KUKA KRL program: MyProgram_338().src

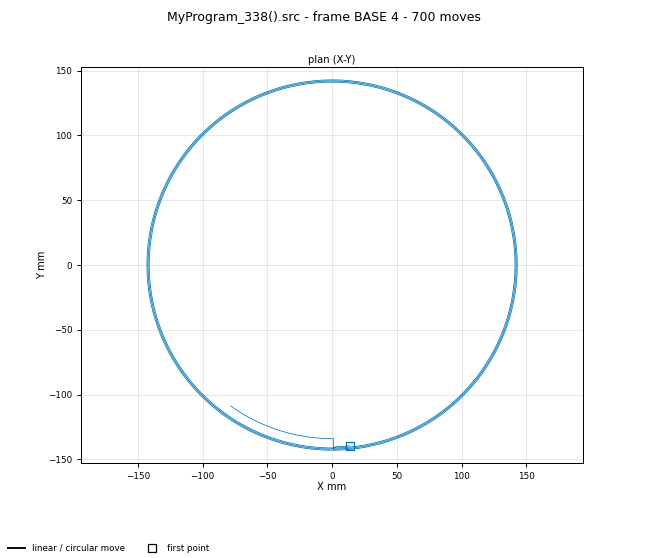
[picture p0: tool path of MyProgram_338().src in frame BASE 4, 700 of 700 moves have a stored position in this frame; points joined in program order, loops and branches not executed]
&ACCESS RVP
&REL 1
&PARAM TEMPLATE = C:\KRC\Roboter\Template\vorgabe
&PARAM EDITMASK = *
DEF MyProgram_338()
; ---- Setting reference (Base) ----
$BASE = BASE_DATA[4]

; --------------------------
; ---- Setting tool (TCP) ----
$TOOL = TOOL_DATA[3]
; --------------------------

$VEL.CP = VEL_APROX_PRINT
Startdeposition()
$VEL.CP = VEL_PRINT
LIN {X 13.5341,Y -139.6097,Z 190,A -74.3045,B 1.205,C 0.2209,E1 1.2499,E2 527.3623} C_DIS
LIN {X 10.5438,Y -139.8677,Z 190,A -75.6606,B 1.2048,C 0.2221,E1 1.246,E2 528.738} C_DIS
LIN {X 6.6617,Y -140.1064,Z 190,A -77.2712,B 1.2046,C 0.223,E1 1.2415,E2 530.3526} C_DIS
LIN {X 2.7568,Y -140.2378,Z 190,A -78.8396,B 1.2045,C 0.2236,E1 1.2371,E2 531.9178} C_DIS
LIN {X 2.7568,Y -140.2378,Z 190,A -78.8396,B 1.2045,C 0.2236,E1 1.2371,E2 531.9178} C_DIS
Enddeposition()
LIN {X 1.0179,Y -141.1573,Z 190,A -79.3498,B 1.2969,C 0.2281,E1 1.3282,E2 532.3992} C_DIS
Startdeposition()
$VEL.CP = VEL_PRINT
LIN {X 4.908,Y -141.079,Z 190,A -77.7249,B 1.297,C 0.2273,E1 1.3328,E2 530.7668} C_DIS
LIN {X 8.6277,Y -140.8992,Z 190,A -76.1602,B 1.2972,C 0.2263,E1 1.3372,E2 529.1935} C_DIS
LIN {X 12.831,Y -140.5802,Z 190,A -74.5145,B 1.2973,C 0.2256,E1 1.3418,E2 527.5564} C_DIS
LIN {X 16.4305,Y -140.2038,Z 190,A -73.2184,B 1.2973,C 0.2254,E1 1.3454,E2 526.2848} C_DIS
LIN {X 19.7873,Y -139.7694,Z 190,A -71.8875,B 1.2975,C 0.2246,E1 1.3491,E2 524.9595} C_DIS
LIN {X 23.0508,Y -139.2683,Z 190,A -70.5385,B 1.2977,C 0.2235,E1 1.3528,E2 523.6084} C_DIS
LIN {X 25.7659,Y -138.7935,Z 190,A -69.2796,B 1.298,C 0.222,E1 1.3564,E2 522.3283} C_DIS
LIN {X 31.931,Y -137.5049,Z 190,A -66.6929,B 1.2984,C 0.2195,E1 1.3635,E2 519.7355} C_DIS
LIN {X 37.4822,Y -136.0967,Z 190,A -64.7983,B 1.2984,C 0.2191,E1 1.3685,E2 517.9024} C_DIS
LIN {X 40.1642,Y -135.3293,Z 190,A -63.2039,B 1.299,C 0.2157,E1 1.3729,E2 516.2395} C_DIS
LIN {X 44.0957,Y -134.0998,Z 190,A -61.9584,B 1.299,C 0.2157,E1 1.3761,E2 515.0555} C_DIS
LIN {X 47.4169,Y -132.9615,Z 190,A -60.616,B 1.2992,C 0.2144,E1 1.3796,E2 513.7243} C_DIS
LIN {X 51.0235,Y -131.6188,Z 190,A -59.1287,B 1.2995,C 0.2128,E1 1.3835,E2 512.2467} C_DIS
LIN {X 54.9963,Y -130.0104,Z 190,A -57.4435,B 1.2998,C 0.2107,E1 1.3879,E2 510.5683} C_DIS
LIN {X 62.0576,Y -126.7908,Z 190,A -54.5002,B 1.3004,C 0.2072,E1 1.3953,E2 507.653} C_DIS
LIN {X 64.5696,Y -125.5308,Z 190,A -52.8888,B 1.301,C 0.2031,E1 1.3995,E2 505.9721} C_DIS
LIN {X 69.0352,Y -123.1325,Z 190,A -51.4052,B 1.3011,C 0.2027,E1 1.4029,E2 504.5708} C_DIS
LIN {X 72.8721,Y -120.9014,Z 190,A -49.7085,B 1.3015,C 0.2003,E1 1.407,E2 502.888} C_DIS
LIN {X 76.531,Y -118.6196,Z 190,A -48.039,B 1.3019,C 0.1977,E1 1.4109,E2 501.2289} C_DIS
LIN {X 80.3918,Y -116.0374,Z 190,A -46.2878,B 1.3023,C 0.195,E1 1.4149,E2 499.4956} C_DIS
LIN {X 84.0888,Y -113.3869,Z 190,A -44.5646,B 1.3027,C 0.1923,E1 1.4188,E2 497.789} C_DIS
LIN {X 87.6501,Y -110.6571,Z 190,A -42.8641,B 1.3031,C 0.1895,E1 1.4225,E2 496.1045} C_DIS
LIN {X 91.1163,Y -107.8213,Z 190,A -41.1614,B 1.3035,C 0.1865,E1 1.4261,E2 494.417} C_DIS
LIN {X 94.5666,Y -104.8082,Z 190,A -39.4314,B 1.304,C 0.1835,E1 1.4297,E2 492.7042} C_DIS
LIN {X 97.9221,Y -101.68,Z 190,A -37.7263,B 1.3044,C 0.1805,E1 1.4332,E2 491.0201} C_DIS
LIN {X 101.0004,Y -98.6228,Z 190,A -36.1083,B 1.3048,C 0.1775,E1 1.4363,E2 489.4213} C_DIS
LIN {X 104.054,Y -95.3951,Z 190,A -34.4823,B 1.3052,C 0.1746,E1 1.4394,E2 487.8192} C_DIS
LIN {X 106.9525,Y -92.1336,Z 190,A -32.8039,B 1.3056,C 0.1712,E1 1.4424,E2 486.1526} C_DIS
LIN {X 110.0028,Y -88.4696,Z 190,A -31.0391,B 1.3061,C 0.1677,E1 1.4455,E2 484.4107} C_DIS
LIN {X 112.8445,Y -84.8153,Z 190,A -29.3426,B 1.3065,C 0.1644,E1 1.4484,E2 482.7386} C_DIS
LIN {X 115.4716,Y -81.2022,Z 190,A -27.6775,B 1.3069,C 0.161,E1 1.451,E2 481.0931} C_DIS
LIN {X 117.9569,Y -77.5475,Z 190,A -25.997,B 1.3074,C 0.1573,E1 1.4536,E2 479.4272} C_DIS
LIN {X 122.4764,Y -70.193,Z 190,A -23.0665,B 1.308,C 0.1521,E1 1.4578,E2 476.575} C_DIS
LIN {X 124.2959,Y -66.9178,Z 190,A -21.3246,B 1.3086,C 0.1469,E1 1.4602,E2 474.8009} C_DIS
LIN {X 126.2627,Y -63.1282,Z 190,A -19.3866,B 1.3092,C 0.1413,E1 1.4626,E2 472.8327} C_DIS
LIN {X 128.4203,Y -58.6139,Z 190,A -17.927,B 1.3094,C 0.1395,E1 1.4642,E2 471.4519} C_DIS
LIN {X 129.9623,Y -55.1114,Z 190,A -16.5262,B 1.3097,C 0.1364,E1 1.4658,E2 470.0713} C_DIS
LIN {X 131.4444,Y -51.4721,Z 190,A -15.3057,B 1.3099,C 0.1345,E1 1.467,E2 468.9016} C_DIS
LIN {X 132.676,Y -48.2089,Z 190,A -14.0439,B 1.3102,C 0.1317,E1 1.4682,E2 467.6601} C_DIS
LIN {X 134.1158,Y -44.0477,Z 190,A -11.9626,B 1.3109,C 0.125,E1 1.4701,E2 465.5368} C_DIS
LIN {X 135.2678,Y -40.3742,Z 190,A -10.7965,B 1.311,C 0.1233,E1 1.471,E2 464.4246} C_DIS
LIN {X 136.1235,Y -37.3864,Z 190,A -9.4656,B 1.3114,C 0.1194,E1 1.472,E2 463.0832} C_DIS
LIN {X 136.9811,Y -34.1103,Z 190,A -8.5109,B 1.3114,C 0.1183,E1 1.4726,E2 462.1854} C_DIS
LIN {X 137.8608,Y -30.3593,Z 190,A -6.9837,B 1.3118,C 0.1142,E1 1.4735,E2 460.6622} C_DIS
LIN {X 138.5251,Y -27.17,Z 190,A -5.8094,B 1.3121,C 0.1115,E1 1.4742,E2 459.5073} C_DIS
LIN {X 139.2306,Y -23.2769,Z 190,A -4.6133,B 1.3122,C 0.1096,E1 1.4747,E2 458.3659} C_DIS
LIN {X 139.7837,Y -19.6869,Z 190,A -3.0728,B 1.3126,C 0.1051,E1 1.4754,E2 456.8155} C_DIS
LIN {X 140.3231,Y -15.3785,Z 190,A -1.5112,B 1.3129,C 0.1015,E1 1.4759,E2 455.2801} C_DIS
LIN {X 140.6221,Y -12.3552,Z 190,A -0.3436,B 1.3131,C 0.0984,E1 1.4762,E2 454.1206} C_DIS
LIN {X 140.8962,Y -8.6768,Z 190,A 0.8959,B 1.3133,C 0.0959,E1 1.4764,E2 452.915} C_DIS
LIN {X 141.0617,Y -5.3511,Z 190,A 2.2341,B 1.3136,C 0.0922,E1 1.4765,E2 451.5778} C_DIS
LIN {X 141.1597,Y -1.024,Z 190,A 3.7703,B 1.3138,C 0.0886,E1 1.4766,E2 450.0702} C_DIS
LIN {X 141.1445,Y 2.2959,Z 190,A 4.9999,B 1.314,C 0.0856,E1 1.4766,E2 448.8556} C_DIS
LIN {X 141.0255,Y 6.2803,Z 190,A 6.4937,B 1.3143,C 0.0818,E1 1.4764,E2 447.3776} C_DIS
LIN {X 140.808,Y 10.0093,Z 190,A 7.8124,B 1.3144,C 0.0788,E1 1.4762,E2 446.0843} C_DIS
LIN {X 140.52,Y 13.4588,Z 190,A 9.1794,B 1.3147,C 0.0751,E1 1.4759,E2 444.7216} C_DIS
LIN {X 140.0009,Y 18.0775,Z 190,A 10.7845,B 1.3149,C 0.0716,E1 1.4753,E2 443.1528} C_DIS
LIN {X 139.5229,Y 21.4556,Z 190,A 11.9532,B 1.3149,C 0.0691,E1 1.4749,E2 442.012} C_DIS
LIN {X 138.7901,Y 25.784,Z 190,A 13.678,B 1.3152,C 0.0645,E1 1.474,E2 440.2939} C_DIS
LIN {X 138.321,Y 28.1823,Z 190,A 15.3295,B 1.3155,C 0.0578,E1 1.4731,E2 438.5546} C_DIS
LIN {X 136.8984,Y 34.4363,Z 190,A 16.7575,B 1.3155,C 0.0578,E1 1.4722,E2 437.2804} C_DIS
LIN {X 135.2163,Y 40.5475,Z 190,A 19.3688,B 1.3158,C 0.0506,E1 1.4702,E2 434.6633} C_DIS
LIN {X 134.0733,Y 44.1752,Z 190,A 20.7118,B 1.3159,C 0.0476,E1 1.4691,E2 433.3457} C_DIS
LIN {X 132.9113,Y 47.5564,Z 190,A 22.0123,B 1.316,C 0.0446,E1 1.4679,E2 432.0642} C_DIS
LIN {X 131.6579,Y 50.9229,Z 190,A 23.21,B 1.3161,C 0.0423,E1 1.4668,E2 430.8996} C_DIS
LIN {X 130.3296,Y 54.232,Z 190,A 24.6209,B 1.3162,C 0.0387,E1 1.4653,E2 429.4928} C_DIS
LIN {X 129.1247,Y 57.0448,Z 190,A 25.9922,B 1.3163,C 0.0347,E1 1.4637,E2 428.1045} C_DIS
LIN {X 127.7624,Y 60.0367,Z 190,A 27.1031,B 1.3163,C 0.0326,E1 1.4624,E2 427.0221} C_DIS
LIN {X 126.0974,Y 63.4566,Z 190,A 28.4339,B 1.3165,C 0.0298,E1 1.4608,E2 425.718} C_DIS
LIN {X 124.1528,Y 67.1841,Z 190,A 30.0382,B 1.3165,C 0.0261,E1 1.4587,E2 424.1263} C_DIS
LIN {X 122.0248,Y 70.9752,Z 190,A 31.5717,B 1.3165,C 0.023,E1 1.4566,E2 422.6218} C_DIS
LIN {X 119.8046,Y 74.6613,Z 190,A 33.111,B 1.3167,C 0.0199,E1 1.4544,E2 421.1083} C_DIS
LIN {X 116.8635,Y 79.1857,Z 190,A 35.1623,B 1.3167,C 0.0153,E1 1.4513,E2 419.0741} C_DIS
LIN {X 114.375,Y 82.7395,Z 190,A 36.8515,B 1.3167,C 0.0115,E1 1.4486,E2 417.3937} C_DIS
LIN {X 112.1974,Y 85.6691,Z 190,A 38.4648,B 1.3167,C 0.0073,E1 1.4458,E2 415.7635} C_DIS
LIN {X 109.8202,Y 88.6959,Z 190,A 39.6553,B 1.3167,C 0.0058,E1 1.4438,E2 414.6195} C_DIS
LIN {X 106.805,Y 92.3049,Z 190,A 41.4079,B 1.3167,C 0.0023,E1 1.4406,E2 412.8862} C_DIS
LIN {X 103.7447,Y 95.7316,Z 190,A 43.1157,B 1.3168,C -0.001,E1 1.4375,E2 411.1978} C_DIS
LIN {X 100.6997,Y 98.9293,Z 190,A 44.7615,B 1.3168,C -0.0041,E1 1.4343,E2 409.5699} C_DIS
LIN {X 95.9388,Y 103.5534,Z 190,A 47.2297,B 1.3168,C -0.0085,E1 1.4294,E2 407.1295} C_DIS
LIN {X 92.6331,Y 106.5204,Z 190,A 48.9428,B 1.3168,C -0.0117,E1 1.4258,E2 405.4274} C_DIS
LIN {X 89.0531,Y 109.5313,Z 190,A 50.7172,B 1.3168,C -0.0148,E1 1.422,E2 403.6683} C_DIS
LIN {X 85.3934,Y 112.4082,Z 190,A 52.4819,B 1.3167,C -0.0178,E1 1.4181,E2 401.9189} C_DIS
LIN {X 82.8015,Y 114.33,Z 190,A 53.8155,B 1.3167,C -0.0203,E1 1.4151,E2 400.5824} C_DIS
LIN {X 78.7128,Y 117.1832,Z 190,A 55.6072,B 1.3167,C -0.0229,E1 1.411,E2 398.8192} C_DIS
LIN {X 74.8526,Y 119.6855,Z 190,A 57.3616,B 1.3166,C -0.0255,E1 1.4069,E2 397.0786} C_DIS
LIN {X 70.9387,Y 122.0459,Z 190,A 59.0952,B 1.3166,C -0.028,E1 1.4027,E2 395.3599} C_DIS
LIN {X 66.8257,Y 124.3454,Z 190,A 60.8711,B 1.3164,C -0.0305,E1 1.3984,E2 393.6007} C_DIS
LIN {X 62.3646,Y 126.6394,Z 190,A 62.6876,B 1.3164,C -0.0326,E1 1.3939,E2 391.8109} C_DIS
LIN {X 59.4283,Y 128.0437,Z 190,A 64.0461,B 1.3164,C -0.0346,E1 1.3904,E2 390.448} C_DIS
LIN {X 56.0027,Y 129.5784,Z 190,A 65.3197,B 1.3164,C -0.0357,E1 1.3872,E2 389.2048} C_DIS
LIN {X 53.4297,Y 130.6624,Z 190,A 66.6139,B 1.3163,C -0.0379,E1 1.3838,E2 387.8915} C_DIS
LIN {X 49.9777,Y 132.0203,Z 190,A 67.8219,B 1.3163,C -0.0386,E1 1.3808,E2 386.7194} C_DIS
LIN {X 46.7189,Y 133.2085,Z 190,A 69.3649,B 1.3162,C -0.0408,E1 1.3766,E2 385.1605} C_DIS
LIN {X 42.9486,Y 134.4705,Z 190,A 70.8645,B 1.3162,C -0.0422,E1 1.3727,E2 383.6749} C_DIS
LIN {X 34.9658,Y 136.764,Z 190,A 74.0337,B 1.316,C -0.045,E1 1.3642,E2 380.5308} C_DIS
LIN {X 28.4039,Y 138.2759,Z 190,A 76.722,B 1.316,C -0.0473,E1 1.3568,E2 377.8486} C_DIS
LIN {X 23.8659,Y 139.1323,Z 190,A 78.5618,B 1.3159,C -0.0487,E1 1.3517,E2 376.0135} C_DIS
LIN {X 20.457,Y 139.6737,Z 190,A 79.9473,B 1.3159,C -0.0497,E1 1.3479,E2 374.6302} C_DIS
LIN {X 16.6678,Y 140.1755,Z 190,A 81.4005,B 1.3159,C -0.0504,E1 1.3439,E2 373.1891} C_DIS
LIN {X 12.8817,Y 140.5754,Z 190,A 82.9809,B 1.3158,C -0.0514,E1 1.3394,E2 371.6052} C_DIS
LIN {X 9.1158,Y 140.8691,Z 190,A 84.4614,B 1.3158,C -0.052,E1 1.3353,E2 370.1314} C_DIS
LIN {X 5.3899,Y 141.0602,Z 190,A 85.9205,B 1.3158,C -0.0526,E1 1.3312,E2 368.6794} C_DIS
LIN {X 0.9406,Y 141.1601,Z 190,A 87.6325,B 1.3158,C -0.0529,E1 1.3264,E2 366.9792} C_DIS
LIN {X -2.4342,Y 141.1422,Z 190,A 89.0428,B 1.3158,C -0.0535,E1 1.3224,E2 365.5646} C_DIS
LIN {X -6.3851,Y 141.0204,Z 190,A 90.7043,B 1.3157,C -0.054,E1 1.3178,E2 363.8972} C_DIS
LIN {X -10.0893,Y 140.8022,Z 190,A 92.1256,B 1.3157,C -0.054,E1 1.3138,E2 362.4865} C_DIS
LIN {X -13.7127,Y 140.4956,Z 190,A 93.5119,B 1.3157,C -0.0538,E1 1.3099,E2 361.1113} C_DIS
LIN {X -18.6946,Y 139.92,Z 190,A 95.7403,B 1.3157,C -0.0543,E1 1.3037,E2 358.8611} C_DIS
LIN {X -22.8858,Y 139.2958,Z 190,A 97.3654,B 1.3157,C -0.0539,E1 1.2992,E2 357.248} C_DIS
LIN {X -26.4042,Y 138.6715,Z 190,A 98.7757,B 1.3157,C -0.0535,E1 1.2953,E2 355.8431} C_DIS
LIN {X -29.2893,Y 138.0918,Z 190,A 99.9238,B 1.3157,C -0.0531,E1 1.2921,E2 354.7011} C_DIS
LIN {X -32.6185,Y 137.3433,Z 190,A 101.2626,B 1.3157,C -0.0526,E1 1.2885,E2 353.3684} C_DIS
LIN {X -35.8886,Y 136.5254,Z 190,A 102.8458,B 1.3157,C -0.0526,E1 1.2841,E2 351.7605} C_DIS
LIN {X -39.734,Y 135.4553,Z 190,A 104.4293,B 1.3157,C -0.0518,E1 1.2798,E2 350.1822} C_DIS
LIN {X -43.1993,Y 134.3904,Z 190,A 105.9471,B 1.3158,C -0.0511,E1 1.2758,E2 348.6597} C_DIS
LIN {X -46.6395,Y 133.236,Z 190,A 107.5721,B 1.3158,C -0.0505,E1 1.2714,E2 347.0176} C_DIS
LIN {X -50.5615,Y 131.7984,Z 190,A 109.3108,B 1.3158,C -0.0494,E1 1.2668,E2 345.2747} C_DIS
LIN {X -53.7243,Y 130.5416,Z 190,A 111.0468,B 1.3158,C -0.049,E1 1.2622,E2 343.4974} C_DIS
LIN {X -57.3028,Y 129.0093,Z 190,A 112.2266,B 1.316,C -0.047,E1 1.2593,E2 342.366} C_DIS
LIN {X -59.9373,Y 127.8083,Z 190,A 113.6246,B 1.316,C -0.0463,E1 1.2556,E2 340.9422} C_DIS
LIN {X -64.8037,Y 125.4116,Z 190,A 115.9255,B 1.316,C -0.0443,E1 1.2498,E2 338.6309} C_DIS
LIN {X -67.7197,Y 123.8608,Z 190,A 117.7515,B 1.316,C -0.0436,E1 1.2452,E2 336.7476} C_DIS
LIN {X -71.9505,Y 121.4525,Z 190,A 119.3362,B 1.3162,C -0.0408,E1 1.2415,E2 335.211} C_DIS
LIN {X -75.8036,Y 119.0856,Z 190,A 121.2722,B 1.3162,C -0.0387,E1 1.2368,E2 333.2641} C_DIS
LIN {X -79.6526,Y 116.546,Z 190,A 123.5288,B 1.3162,C -0.0367,E1 1.2315,E2 330.9625} C_DIS
LIN {X -82.7587,Y 114.3611,Z 190,A 124.8474,B 1.3164,C -0.0342,E1 1.2285,E2 329.6716} C_DIS
LIN {X -86.376,Y 111.6541,Z 190,A 126.7754,B 1.3164,C -0.0316,E1 1.2242,E2 327.7335} C_DIS
LIN {X -89.8002,Y 108.9195,Z 190,A 128.7223,B 1.3164,C -0.0291,E1 1.2199,E2 325.7674} C_DIS
LIN {X -93.1849,Y 106.0386,Z 190,A 130.6176,B 1.3165,C -0.0262,E1 1.2159,E2 323.8623} C_DIS
LIN {X -96.4858,Y 103.044,Z 190,A 132.5822,B 1.3165,C -0.0233,E1 1.2118,E2 321.8801} C_DIS
LIN {X -99.7331,Y 99.9042,Z 190,A 134.5085,B 1.3166,C -0.0201,E1 1.2079,E2 319.9437} C_DIS
LIN {X -102.9011,Y 96.638,Z 190,A 136.4852,B 1.3166,C -0.0167,E1 1.2041,E2 317.9524} C_DIS
LIN {X -105.9155,Y 93.3241,Z 190,A 138.4781,B 1.3167,C -0.0133,E1 1.2003,E2 315.9393} C_DIS
LIN {X -108.8289,Y 89.9095,Z 190,A 140.4573,B 1.3167,C -0.0098,E1 1.1967,E2 313.9421} C_DIS
LIN {X -111.7395,Y 86.2659,Z 190,A 143.0809,B 1.3167,C -0.0062,E1 1.192,E2 311.2295} C_DIS
LIN {X -114.7384,Y 82.2348,Z 190,A 144.6586,B 1.3167,C -0.0017,E1 1.1895,E2 309.7105} C_DIS
LIN {X -117.6216,Y 78.0561,Z 190,A 147.0126,B 1.3167,C 0.0028,E1 1.1858,E2 307.3215} C_DIS
LIN {X -120.0757,Y 74.2256,Z 190,A 148.7681,B 1.3167,C 0.007,E1 1.1832,E2 305.5786} C_DIS
LIN {X -123.2314,Y 68.8593,Z 190,A 151.8354,B 1.3167,C 0.0127,E1 1.1788,E2 302.4458} C_DIS
LIN {X -125.2646,Y 65.0847,Z 190,A 153.7672,B 1.3167,C 0.0169,E1 1.1762,E2 300.4911} C_DIS
LIN {X -126.6424,Y 62.3585,Z 190,A 155.2188,B 1.3167,C 0.0199,E1 1.1744,E2 299.0137} C_DIS
LIN {X -129.065,Y 57.1782,Z 190,A 157.6089,B 1.3166,C 0.0256,E1 1.1716,E2 296.6165} C_DIS
LIN {X -130.8328,Y 53.0067,Z 190,A 159.3647,B 1.3165,C 0.0303,E1 1.1697,E2 294.8724} C_DIS
LIN {X -131.8984,Y 50.3033,Z 190,A 160.9161,B 1.3164,C 0.0333,E1 1.1681,E2 293.2748} C_DIS
LIN {X -133.1199,Y 46.9745,Z 190,A 162.7751,B 1.3163,C 0.037,E1 1.1663,E2 291.3631} C_DIS
LIN {X -134.4319,Y 43.0697,Z 190,A 164.4152,B 1.3161,C 0.0414,E1 1.1649,E2 289.7282} C_DIS
LIN {X -135.4564,Y 39.7301,Z 190,A 165.9508,B 1.3161,C 0.0452,E1 1.1636,E2 288.1785} C_DIS
LIN {X -136.582,Y 35.6764,Z 190,A 168.361,B 1.3159,C 0.0498,E1 1.1619,E2 285.6788} C_DIS
LIN {X -137.5372,Y 31.7898,Z 190,A 169.4919,B 1.3157,C 0.0542,E1 1.1612,E2 284.6128} C_DIS
LIN {X -138.4909,Y 27.3475,Z 190,A 171.9077,B 1.3155,C 0.0593,E1 1.1598,E2 282.1242} C_DIS
LIN {X -139.6177,Y 20.8352,Z 190,A 174.7523,B 1.3151,C 0.0667,E1 1.1584,E2 279.2601} C_DIS
LIN {X -140.2076,Y 16.3991,Z 190,A 176.7981,B 1.3148,C 0.0717,E1 1.1577,E2 277.1855} C_DIS
LIN {X -140.6293,Y 12.2697,Z 190,A 178.8072,B 1.3146,C 0.0765,E1 1.1572,E2 275.1348} C_DIS
LIN {X -141.076,Y 4.9862,Z 190,A -177.8479,B 1.3141,C 0.0848,E1 1.1567,E2 271.741} C_DIS
LIN {X -141.1544,Y -1.6978,Z 190,A -174.8323,B 1.3136,C 0.0924,E1 1.1567,E2 268.6868} C_DIS
LIN {X -141.0591,Y -5.4195,Z 190,A -172.7178,B 1.3132,C 0.0967,E1 1.1569,E2 266.4921} C_DIS
LIN {X -140.8261,Y -9.7619,Z 190,A -171.0856,B 1.3129,C 0.1016,E1 1.1572,E2 264.8788} C_DIS
LIN {X -140.2692,Y -15.8789,Z 190,A -168.3398,B 1.3123,C 0.1085,E1 1.158,E2 262.1004} C_DIS
LIN {X -139.8928,Y -18.9028,Z 190,A -166.9558,B 1.312,C 0.1119,E1 1.1585,E2 260.6971} C_DIS
LIN {X -139.0067,Y -24.5802,Z 190,A -164.4943,B 1.3115,C 0.1183,E1 1.1596,E2 258.2192} C_DIS
LIN {X -138.3734,Y -27.9252,Z 190,A -162.8143,B 1.3111,C 0.1221,E1 1.1605,E2 256.4992} C_DIS
LIN {X -137.3606,Y -32.5471,Z 190,A -160.668,B 1.3106,C 0.1273,E1 1.1619,E2 254.323} C_DIS
LIN {X -136.4058,Y -36.3372,Z 190,A -158.9309,B 1.3102,C 0.1315,E1 1.1631,E2 252.5659} C_DIS
LIN {X -135.1679,Y -40.7057,Z 190,A -156.8508,B 1.3097,C 0.1363,E1 1.1648,E2 250.4541} C_DIS
LIN {X -134.1042,Y -44.0825,Z 190,A -154.8659,B 1.3093,C 0.14,E1 1.1666,E2 248.3939} C_DIS
LIN {X -132.7877,Y -47.8992,Z 190,A -153.742,B 1.3089,C 0.1443,E1 1.1675,E2 247.342} C_DIS
LIN {X -131.7292,Y -50.7396,Z 190,A -152.1032,B 1.3085,C 0.1474,E1 1.1692,E2 245.6471} C_DIS
LIN {X -130.5921,Y -53.6035,Z 190,A -150.7696,B 1.3082,C 0.1505,E1 1.1706,E2 244.3026} C_DIS
LIN {X -128.8207,Y -57.7245,Z 190,A -148.7726,B 1.3077,C 0.155,E1 1.1729,E2 242.2815} C_DIS
LIN {X -127.435,Y -60.7225,Z 190,A -147.3619,B 1.3073,C 0.1582,E1 1.1746,E2 240.8615} C_DIS
LIN {X -125.9601,Y -63.7262,Z 190,A -145.8785,B 1.3069,C 0.1614,E1 1.1764,E2 239.361} C_DIS
LIN {X -124.2033,Y -67.09,Z 190,A -143.9513,B 1.3064,C 0.1649,E1 1.179,E2 237.3801} C_DIS
LIN {X -121.931,Y -71.1369,Z 190,A -141.8664,B 1.3059,C 0.1691,E1 1.182,E2 235.2673} C_DIS
LIN {X -119.8587,Y -74.5743,Z 190,A -140.054,B 1.3054,C 0.1727,E1 1.1847,E2 233.4295} C_DIS
LIN {X -117.3954,Y -78.3949,Z 190,A -138.1225,B 1.3049,C 0.1767,E1 1.1877,E2 231.4861} C_DIS
LIN {X -114.4747,Y -82.6019,Z 190,A -134.7109,B 1.3044,C 0.18,E1 1.1936,E2 227.8842} C_DIS
LIN {X -109.6249,Y -88.9381,Z 190,A -132.2906,B 1.3034,C 0.1873,E1 1.1976,E2 225.5822} C_DIS
LIN {X -105.789,Y -93.4672,Z 190,A -129.7053,B 1.3028,C 0.1918,E1 1.2024,E2 222.972} C_DIS
LIN {X -102.6039,Y -96.9531,Z 190,A -127.6749,B 1.3022,C 0.1952,E1 1.2063,E2 220.9255} C_DIS
LIN {X -96.4816,Y -103.048,Z 190,A -123.8603,B 1.3014,C 0.201,E1 1.214,E2 217.0669} C_DIS
LIN {X -93.118,Y -106.0973,Z 190,A -121.6916,B 1.301,C 0.2035,E1 1.2186,E2 214.8512} C_DIS
LIN {X -90.5663,Y -108.2831,Z 190,A -120.4872,B 1.3006,C 0.2059,E1 1.2212,E2 213.6699} C_DIS
LIN {X -87.1425,Y -111.0568,Z 190,A -118.5675,B 1.3002,C 0.2084,E1 1.2254,E2 211.7311} C_DIS
LIN {X -82.0556,Y -114.8665,Z 190,A -116.0908,B 1.2996,C 0.2122,E1 1.231,E2 209.2693} C_DIS
LIN {X -79.2497,Y -116.8201,Z 190,A -114.3501,B 1.2994,C 0.2134,E1 1.2351,E2 207.4773} C_DIS
LIN {X -75.223,Y -119.4527,Z 190,A -112.3535,B 1.299,C 0.2157,E1 1.2399,E2 205.4741} C_DIS
LIN {X -71.3526,Y -121.8042,Z 190,A -110.4035,B 1.2987,C 0.2176,E1 1.2446,E2 203.5075} C_DIS
LIN {X -67.4815,Y -123.9908,Z 190,A -108.3223,B 1.2985,C 0.2189,E1 1.2498,E2 201.3856} C_DIS
LIN {X -64.6281,Y -125.501,Z 190,A -107.1485,B 1.2982,C 0.2205,E1 1.2527,E2 200.2316} C_DIS
LIN {X -60.5539,Y -127.5155,Z 190,A -105.2903,B 1.2979,C 0.2221,E1 1.2574,E2 198.3711} C_DIS
LIN {X -56.7193,Y -129.2686,Z 190,A -103.4054,B 1.2978,C 0.2231,E1 1.2623,E2 196.4605} C_DIS
LIN {X -53.0407,Y -130.8191,Z 190,A -102.0121,B 1.2975,C 0.2249,E1 1.2659,E2 195.0999} C_DIS
LIN {X -49.836,Y -132.0734,Z 190,A -100.4381,B 1.2974,C 0.2254,E1 1.2701,E2 193.4997} C_DIS
LIN {X -46.557,Y -133.2646,Z 190,A -98.8487,B 1.2974,C 0.2258,E1 1.2743,E2 191.8844} C_DIS
LIN {X -39.2179,Y -135.6064,Z 190,A -95.6814,B 1.2971,C 0.2272,E1 1.2829,E2 188.7103} C_DIS
LIN {X -35.5749,Y -136.6091,Z 190,A -93.8789,B 1.2971,C 0.227,E1 1.2879,E2 186.8677} C_DIS
LIN {X -31.9044,Y -137.511,Z 190,A -92.6406,B 1.2969,C 0.2283,E1 1.2912,E2 185.6724} C_DIS
LIN {X -28.3517,Y -138.2866,Z 190,A -91.1787,B 1.2968,C 0.2287,E1 1.2952,E2 184.212} C_DIS
LIN {X -25.1026,Y -138.9132,Z 190,A -89.8389,B 1.2968,C 0.2289,E1 1.2989,E2 182.8722} C_DIS
LIN {X -21.6302,Y -139.4959,Z 190,A -88.5289,B 1.2967,C 0.2294,E1 1.3025,E2 181.5791} C_DIS
LIN {X -18.6632,Y -139.9242,Z 190,A -87.1996,B 1.2967,C 0.2291,E1 1.3062,E2 180.2328} C_DIS
LIN {X -14.6571,Y -140.4007,Z 190,A -85.4648,B 1.2967,C 0.2287,E1 1.3111,E2 178.483} C_DIS
LIN {X -10.3233,Y -140.7851,Z 190,A -83.8896,B 1.2967,C 0.2292,E1 1.3155,E2 176.9349} C_DIS
LIN {X -6.9557,Y -140.9917,Z 190,A -82.4526,B 1.2967,C 0.2287,E1 1.3195,E2 175.4874} C_DIS
LIN {X -2.8925,Y -141.1346,Z 190,A -80.7503,B 1.2969,C 0.228,E1 1.3243,E2 173.7766} C_DIS
LIN {X 1.0179,Y -141.1573,Z 190,A -79.3471,B 1.2969,C 0.2282,E1 1.3282,E2 172.3996} C_DIS
Enddeposition()
LIN {X 1.0179,Y -141.1573,Z 190,A -79.3471,B 1.2969,C 0.2282,E1 1.3282,E2 172.3996} C_DIS
Startdeposition()
$VEL.CP = VEL_PRINT
LIN {X -1.1496,Y -142.0579,Z 190,A -80.7182,B 1.2965,C 0.2309,E1 1.3242,E2 173.8709} C_DIS
LIN {X -5.1783,Y -141.968,Z 190,A -82.4266,B 1.2964,C 0.2317,E1 1.3193,E2 175.5922} C_DIS
LIN {X -9.748,Y -141.7284,Z 190,A -84.0734,B 1.2964,C 0.2313,E1 1.3148,E2 177.2107} C_DIS
LIN {X -13.0043,Y -141.4666,Z 190,A -85.5689,B 1.2964,C 0.2321,E1 1.3105,E2 178.733} C_DIS
LIN {X -16.9805,Y -141.0435,Z 190,A -87.0493,B 1.2964,C 0.2317,E1 1.3064,E2 180.1946} C_DIS
LIN {X -20.6841,Y -140.5492,Z 190,A -88.5678,B 1.2964,C 0.2317,E1 1.3022,E2 181.7155} C_DIS
LIN {X -24.3142,Y -139.9675,Z 190,A -90.2093,B 1.2964,C 0.232,E1 1.2976,E2 183.381} C_DIS
LIN {X -28.5545,Y -139.1626,Z 190,A -91.8549,B 1.2964,C 0.2314,E1 1.2931,E2 185.0132} C_DIS
LIN {X -31.8541,Y -138.4445,Z 190,A -93.1511,B 1.2965,C 0.2308,E1 1.2895,E2 186.3002} C_DIS
LIN {X -35.0471,Y -137.6707,Z 190,A -94.5933,B 1.2965,C 0.2307,E1 1.2856,E2 187.7601} C_DIS
LIN {X -39.2393,Y -136.5367,Z 190,A -96.2704,B 1.2967,C 0.2298,E1 1.281,E2 189.4268} C_DIS
LIN {X -41.7543,Y -135.787,Z 190,A -97.4715,B 1.2967,C 0.2297,E1 1.2778,E2 190.6492} C_DIS
LIN {X -47.3057,Y -133.9564,Z 190,A -99.8118,B 1.297,C 0.2283,E1 1.2715,E2 192.9878} C_DIS
LIN {X -50.2257,Y -132.8873,Z 190,A -101.1377,B 1.297,C 0.2277,E1 1.268,E2 194.3244} C_DIS
LIN {X -54.5046,Y -131.1899,Z 190,A -103.1165,B 1.2973,C 0.2266,E1 1.2628,E2 196.3215} C_DIS
LIN {X -58.4243,Y -129.4924,Z 190,A -104.8071,B 1.2975,C 0.2251,E1 1.2585,E2 198.0079} C_DIS
LIN {X -61.501,Y -128.0592,Z 190,A -106.2195,B 1.2977,C 0.224,E1 1.2549,E2 199.4269} C_DIS
LIN {X -64.7664,Y -126.4393,Z 190,A -107.745,B 1.2979,C 0.2228,E1 1.251,E2 200.9607} C_DIS
LIN {X -68.2574,Y -124.5914,Z 190,A -109.4754,B 1.2982,C 0.2214,E1 1.2467,E2 202.7113} C_DIS
LIN {X -72.2557,Y -122.3162,Z 190,A -111.4201,B 1.2985,C 0.2195,E1 1.2419,E2 204.6693} C_DIS
LIN {X -76.1205,Y -119.9492,Z 190,A -113.3207,B 1.2988,C 0.2175,E1 1.2374,E2 206.5807} C_DIS
LIN {X -79.8993,Y -117.4659,Z 190,A -115.3075,B 1.2992,C 0.2155,E1 1.2327,E2 208.5913} C_DIS
LIN {X -83.6692,Y -114.8113,Z 190,A -117.3305,B 1.2995,C 0.2132,E1 1.228,E2 210.6381} C_DIS
LIN {X -86.648,Y -112.5803,Z 190,A -118.8516,B 1.2999,C 0.2111,E1 1.2246,E2 212.1621} C_DIS
LIN {X -90.2767,Y -109.692,Z 190,A -120.8277,B 1.3003,C 0.2084,E1 1.2202,E2 214.1535} C_DIS
LIN {X -92.9319,Y -107.4512,Z 190,A -122.2922,B 1.3007,C 0.2063,E1 1.2171,E2 215.6271} C_DIS
LIN {X -96.3953,Y -104.3556,Z 190,A -124.323,B 1.3011,C 0.2034,E1 1.2128,E2 217.6804} C_DIS
LIN {X -99.5095,Y -101.3898,Z 190,A -126.3268,B 1.3015,C 0.2007,E1 1.2087,E2 219.7227} C_DIS
LIN {X -103.2802,Y -97.5461,Z 190,A -128.5035,B 1.3021,C 0.1968,E1 1.2045,E2 221.8999} C_DIS
LIN {X -106.4808,Y -94.0418,Z 190,A -130.6034,B 1.3026,C 0.1934,E1 1.2005,E2 224.0262} C_DIS
LIN {X -108.8941,Y -91.2366,Z 190,A -132.1291,B 1.3031,C 0.1905,E1 1.1977,E2 225.5563} C_DIS
LIN {X -111.4814,Y -88.0572,Z 190,A -133.9903,B 1.3035,C 0.1873,E1 1.1944,E2 227.4469} C_DIS
LIN {X -115.1699,Y -83.1743,Z 190,A -136.4044,B 1.3042,C 0.1822,E1 1.1904,E2 229.8529} C_DIS
LIN {X -117.0664,Y -80.4829,Z 190,A -138.0871,B 1.3046,C 0.1796,E1 1.1876,E2 231.5856} C_DIS
LIN {X -119.1073,Y -77.4305,Z 190,A -140.0407,B 1.305,C 0.1766,E1 1.1845,E2 233.6054} C_DIS
LIN {X -121.1645,Y -74.1702,Z 190,A -141.2379,B 1.3055,C 0.1729,E1 1.1828,E2 234.7519} C_DIS
LIN {X -122.9014,Y -71.255,Z 190,A -142.9111,B 1.3059,C 0.1699,E1 1.1804,E2 236.4676} C_DIS
LIN {X -125.065,Y -67.3856,Z 190,A -144.8827,B 1.3064,C 0.1658,E1 1.1777,E2 238.4644} C_DIS
LIN {X -126.7751,Y -64.1066,Z 190,A -146.4973,B 1.3069,C 0.1623,E1 1.1756,E2 240.0957} C_DIS
LIN {X -129.0309,Y -59.4351,Z 190,A -149.2823,B 1.3075,C 0.1575,E1 1.1722,E2 242.9762} C_DIS
LIN {X -130.8366,Y -55.3505,Z 190,A -150.6671,B 1.308,C 0.1528,E1 1.1707,E2 244.3027} C_DIS
LIN {X -131.9483,Y -52.6438,Z 190,A -152.2078,B 1.3083,C 0.15,E1 1.1691,E2 245.8929} C_DIS
LIN {X -133.3024,Y -49.1174,Z 190,A -153.7449,B 1.3088,C 0.1461,E1 1.1676,E2 247.4314} C_DIS
LIN {X -134.2463,Y -46.4696,Z 190,A -155.0726,B 1.3091,C 0.1432,E1 1.1663,E2 248.7853} C_DIS
LIN {X -135.4703,Y -42.7728,Z 190,A -156.7412,B 1.3095,C 0.1391,E1 1.1648,E2 250.4668} C_DIS
LIN {X -136.4373,Y -39.579,Z 190,A -158.2321,B 1.3099,C 0.1356,E1 1.1636,E2 251.9771} C_DIS
LIN {X -137.2762,Y -36.5619,Z 190,A -159.7143,B 1.3103,C 0.1322,E1 1.1625,E2 253.4886} C_DIS
LIN {X -138.1924,Y -32.9323,Z 190,A -161.4532,B 1.3107,C 0.1282,E1 1.1614,E2 255.2581} C_DIS
LIN {X -139.6734,Y -25.9504,Z 190,A -165.4963,B 1.3114,C 0.1204,E1 1.1591,E2 259.4568} C_DIS
LIN {X -140.672,Y -19.825,Z 190,A -167.3861,B 1.312,C 0.1135,E1 1.1584,E2 261.263} C_DIS
LIN {X -141.1693,Y -15.9162,Z 190,A -169.1057,B 1.3124,C 0.1091,E1 1.1578,E2 262.9994} C_DIS
LIN {X -141.415,Y -13.5418,Z 190,A -170.3144,B 1.3126,C 0.1064,E1 1.1574,E2 264.2406} C_DIS
LIN {X -141.8076,Y -8.5001,Z 190,A -172.5702,B 1.313,C 0.1007,E1 1.157,E2 266.5242} C_DIS
LIN {X -141.9782,Y -4.9187,Z 190,A -174.1063,B 1.3134,C 0.0967,E1 1.1568,E2 268.0715} C_DIS
LIN {X -142.0413,Y -2.4273,Z 190,A -175.3628,B 1.3136,C 0.0938,E1 1.1568,E2 269.3608} C_DIS
LIN {X -142.0359,Y 2.752,Z 190,A -177.6231,B 1.314,C 0.088,E1 1.1568,E2 271.6426} C_DIS
LIN {X -141.9405,Y 5.885,Z 190,A -179.2538,B 1.3142,C 0.0844,E1 1.157,E2 273.3208} C_DIS
LIN {X -141.6628,Y 10.6463,Z 190,A 178.6918,B 1.3145,C 0.079,E1 1.1573,E2 275.3912} C_DIS
LIN {X -141.3323,Y 14.4011,Z 190,A 177.0264,B 1.3148,C 0.0747,E1 1.1578,E2 277.0748} C_DIS
LIN {X -140.8227,Y 18.7245,Z 190,A 175.0749,B 1.3151,C 0.0699,E1 1.1585,E2 279.0506} C_DIS
LIN {X -139.8081,Y 25.2046,Z 190,A 172.1234,B 1.3154,C 0.0625,E1 1.1598,E2 282.0401} C_DIS
LIN {X -138.4993,Y 31.6144,Z 190,A 169.4501,B 1.3157,C 0.0553,E1 1.1614,E2 284.7164} C_DIS
LIN {X -136.9393,Y 37.8067,Z 190,A 166.4817,B 1.316,C 0.0484,E1 1.1634,E2 287.7338} C_DIS
LIN {X -136.1235,Y 40.6506,Z 190,A 164.988,B 1.3161,C 0.0452,E1 1.1646,E2 289.2652} C_DIS
LIN {X -135.1516,Y 43.7705,Z 190,A 163.4252,B 1.3162,C 0.0417,E1 1.166,E2 290.8583} C_DIS
LIN {X -133.9982,Y 47.1851,Z 190,A 161.9202,B 1.3164,C 0.0379,E1 1.1673,E2 292.369} C_DIS
LIN {X -132.6879,Y 50.7543,Z 190,A 160.234,B 1.3164,C 0.0339,E1 1.169,E2 294.0734} C_DIS
LIN {X -131.6998,Y 53.2604,Z 190,A 159.0272,B 1.3165,C 0.0312,E1 1.1703,E2 295.2946} C_DIS
LIN {X -130.1331,Y 56.985,Z 190,A 157.1657,B 1.3166,C 0.0271,E1 1.1724,E2 297.1843} C_DIS
LIN {X -127.2583,Y 63.1418,Z 190,A 154.1319,B 1.3167,C 0.0204,E1 1.176,E2 300.253} C_DIS
LIN {X -125.4752,Y 66.6171,Z 190,A 152.4398,B 1.3168,C 0.0166,E1 1.1782,E2 301.9586} C_DIS
LIN {X -123.2027,Y 70.734,Z 190,A 150.5002,B 1.3168,C 0.0121,E1 1.1809,E2 303.9023} C_DIS
LIN {X -120.6385,Y 75.0226,Z 190,A 148.0173,B 1.3168,C 0.0076,E1 1.1846,E2 306.4418} C_DIS
LIN {X -118.2791,Y 78.6901,Z 190,A 146.1432,B 1.3169,C 0.0037,E1 1.1874,E2 308.3289} C_DIS
LIN {X -115.8515,Y 82.2231,Z 190,A 144.0748,B 1.3169,C 0.0001,E1 1.1908,E2 310.4377} C_DIS
LIN {X -112.796,Y 86.366,Z 190,A 142.1236,B 1.3169,C -0.0044,E1 1.1941,E2 312.3721} C_DIS
LIN {X -110.642,Y 89.1088,Z 190,A 140.4129,B 1.3169,C -0.0071,E1 1.1971,E2 314.119} C_DIS
LIN {X -107.8765,Y 92.4381,Z 190,A 138.4956,B 1.3169,C -0.0105,E1 1.2006,E2 316.056} C_DIS
LIN {X -104.9021,Y 95.8007,Z 190,A 136.4987,B 1.3169,C -0.0138,E1 1.2044,E2 318.0743} C_DIS
LIN {X -101.7567,Y 99.1352,Z 190,A 134.5097,B 1.3168,C -0.0172,E1 1.2083,E2 320.079} C_DIS
LIN {X -98.5698,Y 102.3041,Z 190,A 132.589,B 1.3168,C -0.0203,E1 1.2122,E2 322.0115} C_DIS
LIN {X -95.2915,Y 105.3642,Z 190,A 130.6531,B 1.3168,C -0.0233,E1 1.2162,E2 323.9614} C_DIS
LIN {X -91.9475,Y 108.2944,Z 190,A 128.748,B 1.3166,C -0.0261,E1 1.2203,E2 325.8788} C_DIS
LIN {X -88.5557,Y 111.0852,Z 190,A 126.872,B 1.3166,C -0.0287,E1 1.2244,E2 327.766} C_DIS
LIN {X -85.0461,Y 113.7948,Z 190,A 125.0108,B 1.3166,C -0.0313,E1 1.2286,E2 329.6348} C_DIS
LIN {X -81.5246,Y 116.3439,Z 190,A 123.163,B 1.3165,C -0.0336,E1 1.2328,E2 331.4928} C_DIS
LIN {X -78.3807,Y 118.4846,Z 190,A 121.5246,B 1.3165,C -0.0355,E1 1.2367,E2 333.1425} C_DIS
LIN {X -75.0245,Y 120.6373,Z 190,A 119.8641,B 1.3164,C -0.0374,E1 1.2406,E2 334.8083} C_DIS
LIN {X -71.5323,Y 122.7409,Z 190,A 118.0833,B 1.3164,C -0.0391,E1 1.245,E2 336.6043} C_DIS
LIN {X -67.3017,Y 125.11,Z 190,A 116.0479,B 1.3163,C -0.0411,E1 1.25,E2 338.6479} C_DIS
LIN {X -63.2408,Y 127.2095,Z 190,A 114.0206,B 1.3163,C -0.0427,E1 1.2551,E2 340.6956} C_DIS
LIN {X -58.72,Y 129.3601,Z 190,A 112.1511,B 1.3161,C -0.0447,E1 1.2598,E2 342.5464} C_DIS
LIN {X -56.105,Y 130.5135,Z 190,A 110.8825,B 1.3161,C -0.0455,E1 1.2631,E2 343.8279} C_DIS
LIN {X -52.7535,Y 131.9041,Z 190,A 109.4519,B 1.3161,C -0.0467,E1 1.2668,E2 345.2538} C_DIS
LIN {X -49.4285,Y 133.1859,Z 190,A 107.9084,B 1.3161,C -0.0474,E1 1.2709,E2 346.8091} C_DIS
LIN {X -45.9771,Y 134.417,Z 190,A 106.4448,B 1.3161,C -0.0484,E1 1.2748,E2 348.2703} C_DIS
LIN {X -43.1007,Y 135.3656,Z 190,A 105.1648,B 1.316,C -0.0489,E1 1.2783,E2 349.5563} C_DIS
LIN {X -39.5769,Y 136.4379,Z 190,A 103.6802,B 1.316,C -0.0497,E1 1.2823,E2 351.0401} C_DIS
LIN {X -35.8055,Y 137.4778,Z 190,A 102.0711,B 1.316,C -0.0502,E1 1.2866,E2 352.6522} C_DIS
LIN {X -32.7492,Y 138.2365,Z 190,A 100.7037,B 1.316,C -0.0504,E1 1.2904,E2 354.0302} C_DIS
LIN {X -28.6838,Y 139.1363,Z 190,A 99.2622,B 1.3159,C -0.0515,E1 1.2943,E2 355.443} C_DIS
LIN {X -26.2871,Y 139.609,Z 190,A 98.118,B 1.3159,C -0.0513,E1 1.2975,E2 356.6055} C_DIS
LIN {X -22.3808,Y 140.2893,Z 190,A 96.554,B 1.3159,C -0.0516,E1 1.3018,E2 358.1646} C_DIS
LIN {X -19.6786,Y 140.6929,Z 190,A 95.2372,B 1.3159,C -0.0511,E1 1.3056,E2 359.506} C_DIS
LIN {X -15.4023,Y 141.2246,Z 190,A 93.7328,B 1.3159,C -0.0517,E1 1.3097,E2 360.9822} C_DIS
LIN {X -12.2953,Y 141.5293,Z 190,A 92.3044,B 1.3159,C -0.0512,E1 1.3137,E2 362.43} C_DIS
LIN {X -7.9795,Y 141.8397,Z 190,A 90.6513,B 1.3159,C -0.0512,E1 1.3184,E2 364.0716} C_DIS
LIN {X -4.1639,Y 142.0011,Z 190,A 89.0686,B 1.3159,C -0.0507,E1 1.3228,E2 365.6586} C_DIS
LIN {X -0.6532,Y 142.0606,Z 190,A 87.7263,B 1.3159,C -0.0505,E1 1.3266,E2 366.9917} C_DIS
LIN {X 3.2443,Y 142.0267,Z 190,A 86.2228,B 1.3159,C -0.0501,E1 1.3308,E2 368.4867} C_DIS
LIN {X 6.2401,Y 141.9266,Z 190,A 84.9999,B 1.3159,C -0.0495,E1 1.3342,E2 369.7108} C_DIS
LIN {X 9.1747,Y 141.7661,Z 190,A 83.8408,B 1.3159,C -0.049,E1 1.3375,E2 370.8663} C_DIS
LIN {X 12.2602,Y 141.5322,Z 190,A 82.6139,B 1.316,C -0.0484,E1 1.3409,E2 372.0903} C_DIS
LIN {X 15.8077,Y 141.181,Z 190,A 81.2025,B 1.316,C -0.0476,E1 1.3448,E2 373.4981} C_DIS
LIN {X 19.3167,Y 140.7446,Z 190,A 79.6676,B 1.316,C -0.0463,E1 1.3491,E2 375.0454} C_DIS
LIN {X 23.4979,Y 140.105,Z 190,A 78.0441,B 1.3161,C -0.0453,E1 1.3536,E2 376.6585} C_DIS
LIN {X 27.109,Y 139.4519,Z 190,A 76.7527,B 1.3161,C -0.0447,E1 1.3571,E2 377.9273} C_DIS
LIN {X 29.7541,Y 138.9111,Z 190,A 75.565,B 1.3161,C -0.0434,E1 1.3604,E2 379.1265} C_DIS
LIN {X 33.8151,Y 137.9796,Z 190,A 74.017,B 1.3162,C -0.0423,E1 1.3646,E2 380.6584} C_DIS
LIN {X 36.8127,Y 137.2093,Z 190,A 72.7544,B 1.3162,C -0.041,E1 1.368,E2 381.9224} C_DIS
LIN {X 40.3404,Y 136.2143,Z 190,A 71.0738,B 1.3163,C -0.0386,E1 1.3726,E2 383.6265} C_DIS
LIN {X 44.0074,Y 135.0759,Z 190,A 69.9387,B 1.3163,C -0.0385,E1 1.3755,E2 384.7125} C_DIS
LIN {X 47.1297,Y 134.0174,Z 190,A 68.6827,B 1.3163,C -0.0372,E1 1.3789,E2 385.9594} C_DIS
LIN {X 50.042,Y 132.9561,Z 190,A 67.4439,B 1.3164,C -0.0357,E1 1.3821,E2 387.1966} C_DIS
LIN {X 54.1034,Y 131.3574,Z 190,A 65.8028,B 1.3164,C -0.0339,E1 1.3864,E2 388.8232} C_DIS
LIN {X 57.0871,Y 130.0889,Z 190,A 64.5512,B 1.3165,C -0.0323,E1 1.3896,E2 390.068} C_DIS
LIN {X 59.9371,Y 128.7987,Z 190,A 63.3161,B 1.3165,C -0.0306,E1 1.3927,E2 391.2996} C_DIS
LIN {X 64.0593,Y 126.7992,Z 190,A 61.5274,B 1.3166,C -0.0281,E1 1.3972,E2 393.081} C_DIS
LIN {X 67.7379,Y 124.8748,Z 190,A 59.9115,B 1.3166,C -0.0258,E1 1.4012,E2 394.6898} C_DIS
LIN {X 71.8465,Y 122.5566,Z 190,A 58.198,B 1.3166,C -0.0235,E1 1.4053,E2 396.3804} C_DIS
LIN {X 75.0768,Y 120.6048,Z 190,A 56.7116,B 1.3167,C -0.0211,E1 1.4088,E2 397.8623} C_DIS
LIN {X 78.7534,Y 118.2369,Z 190,A 55.1972,B 1.3167,C -0.0192,E1 1.4123,E2 399.3465} C_DIS
LIN {X 82.0273,Y 115.9896,Z 190,A 53.6191,B 1.3168,C -0.0164,E1 1.4159,E2 400.9218} C_DIS
LIN {X 85.0452,Y 113.7955,Z 190,A 52.2059,B 1.3168,C -0.0141,E1 1.4191,E2 402.3239} C_DIS
LIN {X 88.3846,Y 111.2214,Z 190,A 50.6093,B 1.3168,C -0.0113,E1 1.4226,E2 403.9078} C_DIS
LIN {X 91.5838,Y 108.6027,Z 190,A 49.075,B 1.3168,C -0.0087,E1 1.4259,E2 405.426} C_DIS
LIN {X 94.6364,Y 105.9529,Z 190,A 47.5519,B 1.3168,C -0.006,E1 1.4291,E2 406.936} C_DIS
LIN {X 97.7531,Y 103.0849,Z 190,A 45.8624,B 1.3169,C -0.0025,E1 1.4325,E2 408.6233} C_DIS
LIN {X 100.5029,Y 100.4059,Z 190,A 44.4785,B 1.3169,C -0.0001,E1 1.4352,E2 409.9871} C_DIS
LIN {X 103.7485,Y 97.0483,Z 190,A 42.7679,B 1.3169,C 0.0031,E1 1.4385,E2 411.6766} C_DIS
LIN {X 106.6504,Y 93.85,Z 190,A 41.2239,B 1.3169,C 0.0059,E1 1.4413,E2 413.1964} C_DIS
LIN {X 109.2614,Y 90.7966,Z 190,A 39.7193,B 1.3169,C 0.009,E1 1.444,E2 414.6869} C_DIS
LIN {X 111.7886,Y 87.6661,Z 190,A 38.1863,B 1.3169,C 0.0122,E1 1.4467,E2 416.209} C_DIS
LIN {X 114.5949,Y 83.9647,Z 190,A 36.4939,B 1.3169,C 0.0156,E1 1.4495,E2 417.8792} C_DIS
LIN {X 117.1185,Y 80.4069,Z 190,A 34.8751,B 1.3168,C 0.0191,E1 1.452,E2 419.4807} C_DIS
LIN {X 119.6719,Y 76.5549,Z 190,A 33.2888,B 1.3168,C 0.022,E1 1.4544,E2 421.0325} C_DIS
LIN {X 121.6958,Y 73.2955,Z 190,A 31.7429,B 1.3167,C 0.0259,E1 1.4567,E2 422.5787} C_DIS
LIN {X 123.9564,Y 69.404,Z 190,A 30.0935,B 1.3166,C 0.0295,E1 1.4589,E2 424.2076} C_DIS
LIN {X 126.1196,Y 65.3899,Z 190,A 28.4724,B 1.3165,C 0.0329,E1 1.461,E2 425.8015} C_DIS
LIN {X 127.7573,Y 62.1302,Z 190,A 27.1479,B 1.3165,C 0.0358,E1 1.4626,E2 427.1078} C_DIS
LIN {X 129.0983,Y 59.2893,Z 190,A 25.9665,B 1.3163,C 0.0386,E1 1.464,E2 428.2786} C_DIS
LIN {X 130.5332,Y 56.0595,Z 190,A 24.7114,B 1.3163,C 0.0413,E1 1.4654,E2 429.5124} C_DIS
LIN {X 131.7845,Y 53.0503,Z 190,A 23.4513,B 1.3162,C 0.0444,E1 1.4667,E2 430.7659} C_DIS
LIN {X 133.3538,Y 48.9793,Z 190,A 21.9082,B 1.316,C 0.0478,E1 1.4682,E2 432.2819} C_DIS
LIN {X 134.3249,Y 46.243,Z 190,A 20.8255,B 1.316,C 0.0504,E1 1.4692,E2 433.3536} C_DIS
LIN {X 135.5608,Y 42.4896,Z 190,A 19.1221,B 1.3157,C 0.0554,E1 1.4707,E2 435.0718} C_DIS
LIN {X 136.54,Y 39.2282,Z 190,A 18.1728,B 1.3157,C 0.0566,E1 1.4714,E2 435.9668} C_DIS
LIN {X 137.3638,Y 36.2333,Z 190,A 16.9274,B 1.3155,C 0.0599,E1 1.4723,E2 437.2118} C_DIS
LIN {X 138.437,Y 31.8873,Z 190,A 15.1556,B 1.3153,C 0.0647,E1 1.4734,E2 438.98} C_DIS
LIN {X 139.3452,Y 27.657,Z 190,A 13.6541,B 1.3151,C 0.068,E1 1.4742,E2 440.4506} C_DIS
LIN {X 140.1767,Y 23.0686,Z 190,A 12.0114,B 1.3149,C 0.0718,E1 1.475,E2 442.0629} C_DIS
LIN {X 140.7499,Y 19.2798,Z 190,A 10.7142,B 1.3148,C 0.0745,E1 1.4755,E2 443.3284} C_DIS
LIN {X 141.0888,Y 16.6008,Z 190,A 9.7531,B 1.3147,C 0.0768,E1 1.4758,E2 444.273} C_DIS
LIN {X 141.4156,Y 13.5356,Z 190,A 8.5909,B 1.3145,C 0.0797,E1 1.4761,E2 445.4251} C_DIS
LIN {X 141.7147,Y 9.9358,Z 190,A 7.286,B 1.3143,C 0.0829,E1 1.4764,E2 446.7107} C_DIS
LIN {X 141.8934,Y 6.9222,Z 190,A 6.1834,B 1.3141,C 0.0855,E1 1.4766,E2 447.7987} C_DIS
LIN {X 142.0129,Y 3.7423,Z 190,A 5.0211,B 1.3139,C 0.0884,E1 1.4766,E2 448.9455} C_DIS
LIN {X 142.0625,Y -0.3146,Z 190,A 3.4828,B 1.3137,C 0.0924,E1 1.4767,E2 450.4716} C_DIS
LIN {X 142.0045,Y -4.0431,Z 190,A 2.1804,B 1.3135,C 0.0953,E1 1.4767,E2 451.7478} C_DIS
LIN {X 141.8409,Y -7.9601,Z 190,A 0.6141,B 1.3131,C 0.0996,E1 1.4764,E2 453.3133} C_DIS
LIN {X 141.5765,Y -11.7356,Z 190,A -0.7152,B 1.3129,C 0.1027,E1 1.4761,E2 454.6169} C_DIS
LIN {X 141.1096,Y -16.4261,Z 190,A -2.4266,B 1.3126,C 0.1068,E1 1.4756,E2 456.3039} C_DIS
LIN {X 140.5775,Y -20.486,Z 190,A -3.9544,B 1.3123,C 0.1106,E1 1.4751,E2 457.816} C_DIS
LIN {X 139.982,Y -24.2328,Z 190,A -5.2161,B 1.312,C 0.1132,E1 1.4745,E2 459.0423} C_DIS
LIN {X 139.487,Y -26.9258,Z 190,A -6.1863,B 1.3118,C 0.1154,E1 1.474,E2 459.9949} C_DIS
LIN {X 138.9366,Y -29.6358,Z 190,A -7.1608,B 1.3116,C 0.1176,E1 1.4735,E2 460.9509} C_DIS
LIN {X 138.3205,Y -32.397,Z 190,A -8.4072,B 1.3113,C 0.1214,E1 1.4727,E2 462.2125} C_DIS
LIN {X 137.0674,Y -37.3433,Z 190,A -10.1109,B 1.311,C 0.1248,E1 1.4715,E2 463.8691} C_DIS
LIN {X 136.3075,Y -40.0222,Z 190,A -11.9567,B 1.3102,C 0.1323,E1 1.47,E2 465.8143} C_DIS
LIN {X 134.2569,Y -46.4391,Z 190,A -13.384,B 1.3103,C 0.1316,E1 1.4689,E2 467.0667} C_DIS
LIN {X 132.648,Y -50.8568,Z 190,A -15.2853,B 1.3098,C 0.1367,E1 1.467,E2 468.9701} C_DIS
LIN {X 131.2839,Y -54.2795,Z 190,A -16.7916,B 1.3094,C 0.1407,E1 1.4654,E2 470.4804} C_DIS
LIN {X 129.6292,Y -58.1184,Z 190,A -18.195,B 1.3091,C 0.1434,E1 1.4639,E2 471.8456} C_DIS
LIN {X 127.5683,Y -62.5134,Z 190,A -19.8626,B 1.3087,C 0.1467,E1 1.462,E2 473.4743} C_DIS
LIN {X 125.8274,Y -65.9464,Z 190,A -21.4439,B 1.3082,C 0.1508,E1 1.4599,E2 475.0607} C_DIS
LIN {X 123.8175,Y -69.651,Z 190,A -23.3321,B 1.3076,C 0.1562,E1 1.4573,E2 476.9766} C_DIS
LIN {X 121.8509,Y -73.0374,Z 190,A -24.598,B 1.3074,C 0.1583,E1 1.4556,E2 478.1998} C_DIS
LIN {X 119.9569,Y -76.1083,Z 190,A -25.8389,B 1.3071,C 0.1606,E1 1.4538,E2 479.4118} C_DIS
LIN {X 117.6012,Y -79.6994,Z 190,A -27.4315,B 1.3067,C 0.1639,E1 1.4513,E2 480.9861} C_DIS
LIN {X 114.9904,Y -83.4221,Z 190,A -29.0964,B 1.3062,C 0.1673,E1 1.4487,E2 482.6285} C_DIS
LIN {X 112.3499,Y -86.9456,Z 190,A -30.7462,B 1.3058,C 0.1707,E1 1.4459,E2 484.2618} C_DIS
LIN {X 109.5026,Y -90.5053,Z 190,A -32.4522,B 1.3053,C 0.1741,E1 1.4429,E2 485.9505} C_DIS
LIN {X 106.3725,Y -94.1643,Z 190,A -34.2401,B 1.3049,C 0.1776,E1 1.4397,E2 487.7179} C_DIS
LIN {X 103.214,Y -97.6162,Z 190,A -35.9699,B 1.3044,C 0.1808,E1 1.4364,E2 489.4268} C_DIS
LIN {X 99.9038,Y -101.0018,Z 190,A -37.739,B 1.304,C 0.1841,E1 1.4329,E2 491.1773} C_DIS
LIN {X 96.4945,Y -104.2642,Z 190,A -39.5096,B 1.3035,C 0.1873,E1 1.4294,E2 492.9305} C_DIS
LIN {X 93.0089,Y -107.3849,Z 190,A -41.2728,B 1.3031,C 0.1904,E1 1.4257,E2 494.6774} C_DIS
LIN {X 89.4644,Y -110.3552,Z 190,A -43.0152,B 1.3026,C 0.1934,E1 1.422,E2 496.4036} C_DIS
LIN {X 85.7344,Y -113.277,Z 190,A -44.7592,B 1.3022,C 0.1961,E1 1.4181,E2 498.125} C_DIS
LIN {X 82.3296,Y -115.7756,Z 190,A -46.3665,B 1.3018,C 0.1987,E1 1.4145,E2 499.7198} C_DIS
LIN {X 78.6335,Y -118.3169,Z 190,A -48.0288,B 1.3014,C 0.2012,E1 1.4107,E2 501.3623} C_DIS
LIN {X 74.961,Y -120.6768,Z 190,A -49.7128,B 1.301,C 0.2038,E1 1.4067,E2 503.0365} C_DIS
LIN {X 70.9119,Y -123.1,Z 190,A -51.5226,B 1.3006,C 0.2065,E1 1.4024,E2 504.8343} C_DIS
LIN {X 65.9222,Y -125.8401,Z 190,A -53.6171,B 1.3002,C 0.2091,E1 1.3973,E2 506.9011} C_DIS
LIN {X 62.3025,Y -127.6723,Z 190,A -55.1998,B 1.2999,C 0.2112,E1 1.3933,E2 508.4773} C_DIS
LIN {X 58.2476,Y -129.5714,Z 190,A -57.1834,B 1.2993,C 0.2147,E1 1.3882,E2 510.4879} C_DIS
LIN {X 54.7488,Y -131.0879,Z 190,A -58.3473,B 1.2993,C 0.215,E1 1.3853,E2 511.5985} C_DIS
LIN {X 51.3432,Y -132.4589,Z 190,A -59.7083,B 1.299,C 0.2163,E1 1.3818,E2 512.9431} C_DIS
LIN {X 48.3358,Y -133.5858,Z 190,A -60.9787,B 1.2988,C 0.2178,E1 1.3784,E2 514.2107} C_DIS
LIN {X 44.4695,Y -134.9227,Z 190,A -62.8372,B 1.2983,C 0.2207,E1 1.3734,E2 516.1009} C_DIS
LIN {X 40.9608,Y -136.0299,Z 190,A -63.9284,B 1.2983,C 0.2207,E1 1.3706,E2 517.1358} C_DIS
LIN {X 37.431,Y -137.0443,Z 190,A -65.3616,B 1.2981,C 0.222,E1 1.3668,E2 518.5629} C_DIS
LIN {X 34.3033,Y -137.8595,Z 190,A -66.6946,B 1.2978,C 0.2234,E1 1.3631,E2 519.9011} C_DIS
LIN {X 25.9667,Y -139.6703,Z 190,A -69.9351,B 1.2974,C 0.2256,E1 1.3543,E2 523.1145} C_DIS
LIN {X 22.8819,Y -140.2078,Z 190,A -71.147,B 1.2974,C 0.2264,E1 1.3509,E2 524.3196} C_DIS
LIN {X 19.6762,Y -140.6933,Z 190,A -72.5577,B 1.2971,C 0.2278,E1 1.347,E2 525.7462} C_DIS
LIN {X 15.6321,Y -141.1999,Z 190,A -74.1564,B 1.2969,C 0.2287,E1 1.3425,E2 527.3392} C_DIS
LIN {X 11.802,Y -141.5709,Z 190,A -75.5939,B 1.2969,C 0.2291,E1 1.3385,E2 528.7608} C_DIS
LIN {X 7.4805,Y -141.8653,Z 190,A -77.287,B 1.2967,C 0.2298,E1 1.3338,E2 530.447} C_DIS
LIN {X 4.2105,Y -141.9999,Z 190,A -78.5439,B 1.2967,C 0.2301,E1 1.3303,E2 531.6953} C_DIS
LIN {X 1.0282,Y -142.0561,Z 190,A -79.3363,B 1.2969,C 0.2288,E1 1.3283,E2 532.4159} C_DIS
Enddeposition()
LIN {X 1.0282,Y -142.0561,Z 190,A -79.3365,B 1.2969,C 0.2288,E1 1.3283,E2 532.416} C_DIS
Startdeposition()
$VEL.CP = VEL_PRINT
LIN {X 1.7616,Y -142.9514,Z 190,A -78.9154,B 1.2968,C 0.2288,E1 1.3293,E2 532.0023} C_DIS
LIN {X 5.2668,Y -142.8642,Z 190,A -77.5034,B 1.2968,C 0.2282,E1 1.3333,E2 530.5885} C_DIS
LIN {X 8.7679,Y -142.6917,Z 190,A -76.1725,B 1.2969,C 0.2278,E1 1.337,E2 529.2679} C_DIS
LIN {X 12.2835,Y -142.4323,Z 190,A -74.7749,B 1.2971,C 0.227,E1 1.3409,E2 527.8718} C_DIS
LIN {X 15.9944,Y -142.065,Z 190,A -73.3439,B 1.2971,C 0.2263,E1 1.3449,E2 526.4495} C_DIS
LIN {X 19.2469,Y -141.6608,Z 190,A -72.0619,B 1.2973,C 0.2256,E1 1.3485,E2 525.1714} C_DIS
LIN {X 22.7131,Y -141.1473,Z 190,A -70.6119,B 1.2975,C 0.2243,E1 1.3525,E2 523.7137} C_DIS
LIN {X 26.2114,Y -140.5387,Z 190,A -69.2975,B 1.2977,C 0.2236,E1 1.3561,E2 522.4146} C_DIS
LIN {X 29.6475,Y -139.8537,Z 190,A -67.9426,B 1.2978,C 0.2226,E1 1.3598,E2 521.0662} C_DIS
LIN {X 33.0597,Y -139.0863,Z 190,A -66.592,B 1.298,C 0.2215,E1 1.3635,E2 519.7223} C_DIS
LIN {X 36.4471,Y -138.2371,Z 190,A -65.2455,B 1.2982,C 0.2203,E1 1.3671,E2 518.3828} C_DIS
LIN {X 39.8102,Y -137.3062,Z 190,A -63.8543,B 1.2985,C 0.2189,E1 1.3709,E2 516.9918} C_DIS
LIN {X 43.9179,Y -136.0482,Z 190,A -62.2273,B 1.2987,C 0.2173,E1 1.3752,E2 515.3777} C_DIS
LIN {X 48.3801,Y -134.5253,Z 190,A -60.4948,B 1.299,C 0.2158,E1 1.3798,E2 513.6673} C_DIS
LIN {X 51.4502,Y -133.3818,Z 190,A -59.1917,B 1.2993,C 0.2142,E1 1.3832,E2 512.3647} C_DIS
LIN {X 54.742,Y -132.0649,Z 190,A -57.7945,B 1.2995,C 0.2124,E1 1.3868,E2 510.9701} C_DIS
LIN {X 58.7565,Y -130.3285,Z 190,A -56.0688,B 1.2999,C 0.2101,E1 1.3912,E2 509.2472} C_DIS
LIN {X 62.8154,Y -128.4216,Z 190,A -54.4234,B 1.3002,C 0.2082,E1 1.3953,E2 507.623} C_DIS
LIN {X 65.8362,Y -126.9005,Z 190,A -53.1013,B 1.3005,C 0.2063,E1 1.3986,E2 506.3049} C_DIS
LIN {X 69.7096,Y -124.8157,Z 190,A -51.5082,B 1.3008,C 0.2044,E1 1.4025,E2 504.7356} C_DIS
LIN {X 73.4033,Y -122.6795,Z 190,A -49.8919,B 1.3012,C 0.2021,E1 1.4064,E2 503.1318} C_DIS
LIN {X 76.4857,Y -120.7817,Z 190,A -48.5416,B 1.3015,C 0.2001,E1 1.4096,E2 501.7952} C_DIS
LIN {X 80.0557,Y -118.4455,Z 190,A -46.9371,B 1.3019,C 0.1977,E1 1.4133,E2 500.2049} C_DIS
LIN {X 83.2845,Y -116.1979,Z 190,A -45.3912,B 1.3023,C 0.195,E1 1.4168,E2 498.6623} C_DIS
LIN {X 86.8112,Y -113.5872,Z 190,A -43.7603,B 1.3027,C 0.1923,E1 1.4204,E2 497.0489} C_DIS
LIN {X 90.0149,Y -111.066,Z 190,A -42.3125,B 1.303,C 0.1902,E1 1.4235,E2 495.627} C_DIS
LIN {X 92.7983,Y -108.751,Z 190,A -40.8599,B 1.3034,C 0.1873,E1 1.4266,E2 494.1731} C_DIS
LIN {X 96.0963,Y -105.8477,Z 190,A -39.3541,B 1.3037,C 0.1852,E1 1.4297,E2 492.7031} C_DIS
LIN {X 98.6633,Y -103.4592,Z 190,A -37.9359,B 1.3041,C 0.1822,E1 1.4326,E2 491.282} C_DIS
LIN {X 101.7889,Y -100.3863,Z 190,A -36.2925,B 1.3046,C 0.1791,E1 1.4358,E2 489.6537} C_DIS
LIN {X 104.7395,Y -97.3031,Z 190,A -34.8057,B 1.3049,C 0.1767,E1 1.4386,E2 488.1981} C_DIS
LIN {X 107.1781,Y -94.6103,Z 190,A -33.3612,B 1.3053,C 0.1735,E1 1.4413,E2 486.7541} C_DIS
LIN {X 110.0275,Y -91.2809,Z 190,A -31.8672,B 1.3056,C 0.1711,E1 1.444,E2 485.2967} C_DIS
LIN {X 112.6328,Y -88.0466,Z 190,A -30.3012,B 1.3061,C 0.1678,E1 1.4467,E2 483.7437} C_DIS
LIN {X 115.2871,Y -84.5407,Z 190,A -28.6974,B 1.3065,C 0.1646,E1 1.4493,E2 482.1614} C_DIS
LIN {X 117.4557,Y -81.501,Z 190,A -27.3405,B 1.3068,C 0.1619,E1 1.4515,E2 480.8233} C_DIS
LIN {X 119.7729,Y -78.0561,Z 190,A -25.7988,B 1.3072,C 0.1586,E1 1.4538,E2 479.2979} C_DIS
LIN {X 121.7928,Y -74.865,Z 190,A -24.4362,B 1.3075,C 0.1558,E1 1.4558,E2 477.9558} C_DIS
LIN {X 123.9123,Y -71.3031,Z 190,A -22.9009,B 1.3079,C 0.1524,E1 1.4579,E2 476.4372} C_DIS
LIN {X 125.7282,Y -68.0504,Z 190,A -21.4818,B 1.3083,C 0.1491,E1 1.4598,E2 475.0275} C_DIS
LIN {X 127.3003,Y -65.0564,Z 190,A -20.3208,B 1.3086,C 0.1468,E1 1.4613,E2 473.8932} C_DIS
LIN {X 128.8501,Y -61.9309,Z 190,A -19.039,B 1.3089,C 0.144,E1 1.4629,E2 472.6269} C_DIS
LIN {X 130.3857,Y -58.6285,Z 190,A -17.627,B 1.3093,C 0.1405,E1 1.4645,E2 471.2205} C_DIS
LIN {X 132.1685,Y -54.4939,Z 190,A -16.068,B 1.3096,C 0.1373,E1 1.4661,E2 469.695} C_DIS
LIN {X 133.4648,Y -51.2367,Z 190,A -14.8058,B 1.3099,C 0.1344,E1 1.4674,E2 468.4519} C_DIS
LIN {X 134.6028,Y -48.1652,Z 190,A -13.5925,B 1.3102,C 0.1316,E1 1.4686,E2 467.2516} C_DIS
LIN {X 135.7698,Y -44.771,Z 190,A -12.2967,B 1.3105,C 0.1286,E1 1.4697,E2 465.9748} C_DIS
LIN {X 137.0283,Y -40.7594,Z 190,A -10.7017,B 1.3109,C 0.1246,E1 1.471,E2 464.3914} C_DIS
LIN {X 137.8736,Y -37.8035,Z 190,A -9.6548,B 1.3111,C 0.1224,E1 1.4717,E2 463.3695} C_DIS
LIN {X 138.7365,Y -34.5021,Z 190,A -8.4138,B 1.3114,C 0.1195,E1 1.4726,E2 462.1452} C_DIS
LIN {X 139.5407,Y -31.0917,Z 190,A -7.1437,B 1.3116,C 0.1165,E1 1.4734,E2 460.8929} C_DIS
LIN {X 140.2613,Y -27.6625,Z 190,A -5.8703,B 1.3119,C 0.1134,E1 1.4741,E2 459.6367} C_DIS
LIN {X 140.8965,Y -24.2162,Z 190,A -4.585,B 1.3122,C 0.1103,E1 1.4747,E2 458.367} C_DIS
LIN {X 141.4469,Y -20.7563,Z 190,A -3.3712,B 1.3124,C 0.1076,E1 1.4752,E2 457.1786} C_DIS
LIN {X 141.8877,Y -17.4921,Z 190,A -2.1192,B 1.3126,C 0.1044,E1 1.4756,E2 455.9352} C_DIS
LIN {X 142.2951,Y -13.7803,Z 190,A -0.7739,B 1.3129,C 0.1011,E1 1.476,E2 454.6097} C_DIS
LIN {X 142.5902,Y -10.2882,Z 190,A 0.4607,B 1.3131,C 0.0983,E1 1.4763,E2 453.3976} C_DIS
LIN {X 142.8001,Y -6.7894,Z 190,A 1.7538,B 1.3133,C 0.0951,E1 1.4765,E2 452.1189} C_DIS
LIN {X 142.925,Y -3.2785,Z 190,A 3.0509,B 1.3136,C 0.0918,E1 1.4765,E2 450.8361} C_DIS
LIN {X 142.963,Y -0.0021,Z 190,A 4.3569,B 1.3138,C 0.0882,E1 1.4765,E2 449.5305} C_DIS
LIN {X 142.9185,Y 3.5106,Z 190,A 5.5106,B 1.314,C 0.0858,E1 1.4765,E2 448.4105} C_DIS
LIN {X 142.7774,Y 7.2416,Z 190,A 6.8173,B 1.3142,C 0.0828,E1 1.4764,E2 447.1286} C_DIS
LIN {X 142.5554,Y 10.7652,Z 190,A 8.1029,B 1.3144,C 0.0797,E1 1.4761,E2 445.8598} C_DIS
LIN {X 142.2503,Y 14.2478,Z 190,A 9.3871,B 1.3146,C 0.0765,E1 1.4758,E2 444.5907} C_DIS
LIN {X 141.8593,Y 17.7302,Z 190,A 10.6544,B 1.3147,C 0.0735,E1 1.4754,E2 443.3411} C_DIS
LIN {X 141.4155,Y 20.976,Z 190,A 11.8496,B 1.3149,C 0.0706,E1 1.4749,E2 442.1611} C_DIS
LIN {X 140.8166,Y 24.6722,Z 190,A 13.1593,B 1.315,C 0.0676,E1 1.4743,E2 440.8761} C_DIS
LIN {X 140.209,Y 27.92,Z 190,A 14.4186,B 1.3152,C 0.0643,E1 1.4737,E2 439.6249} C_DIS
LIN {X 139.4846,Y 31.3376,Z 190,A 15.7667,B 1.3154,C 0.0608,E1 1.4729,E2 438.2831} C_DIS
LIN {X 138.6767,Y 34.7374,Z 190,A 16.9528,B 1.3154,C 0.0583,E1 1.4721,E2 437.125} C_DIS
LIN {X 137.7863,Y 38.1156,Z 190,A 18.2206,B 1.3156,C 0.0553,E1 1.4712,E2 435.8741} C_DIS
LIN {X 136.7199,Y 41.7776,Z 190,A 19.5961,B 1.3158,C 0.0521,E1 1.4701,E2 434.5182} C_DIS
LIN {X 135.6738,Y 45.0593,Z 190,A 20.9586,B 1.3158,C 0.0485,E1 1.4689,E2 433.1575} C_DIS
LIN {X 134.0002,Y 49.8171,Z 190,A 22.6934,B 1.316,C 0.0448,E1 1.4673,E2 431.4597} C_DIS
LIN {X 132.739,Y 53.0867,Z 190,A 24.0161,B 1.3161,C 0.0416,E1 1.466,E2 430.1471} C_DIS
LIN {X 131.3069,Y 56.535,Z 190,A 25.2792,B 1.3162,C 0.039,E1 1.4646,E2 428.9141} C_DIS
LIN {X 129.9252,Y 59.6428,Z 190,A 26.5808,B 1.3162,C 0.0358,E1 1.4631,E2 427.62} C_DIS
LIN {X 128.4264,Y 62.8056,Z 190,A 27.8118,B 1.3164,C 0.0332,E1 1.4617,E2 426.4109} C_DIS
LIN {X 126.9034,Y 65.8307,Z 190,A 29.1795,B 1.3164,C 0.0297,E1 1.4599,E2 425.0416} C_DIS
LIN {X 124.8172,Y 69.707,Z 190,A 30.7168,B 1.3165,C 0.0266,E1 1.4579,E2 423.5331} C_DIS
LIN {X 122.6808,Y 73.401,Z 190,A 32.2861,B 1.3165,C 0.0231,E1 1.4557,E2 421.9817} C_DIS
LIN {X 120.3661,Y 77.1379,Z 190,A 33.901,B 1.3166,C 0.0196,E1 1.4533,E2 420.3852} C_DIS
LIN {X 117.9498,Y 80.7843,Z 190,A 35.5113,B 1.3166,C 0.0162,E1 1.4508,E2 418.7928} C_DIS
LIN {X 115.7976,Y 83.8401,Z 190,A 36.9422,B 1.3167,C 0.013,E1 1.4485,E2 417.3702} C_DIS
LIN {X 113.2339,Y 87.2723,Z 190,A 38.4425,B 1.3167,C 0.0102,E1 1.446,E2 415.8972} C_DIS
LIN {X 110.58,Y 90.6108,Z 190,A 40.0118,B 1.3167,C 0.0071,E1 1.4433,E2 414.3455} C_DIS
LIN {X 107.9046,Y 93.7812,Z 190,A 41.5863,B 1.3167,C 0.0038,E1 1.4404,E2 412.7819} C_DIS
LIN {X 104.9319,Y 97.0965,Z 190,A 43.2485,B 1.3167,C 0.0005,E1 1.4373,E2 411.1351} C_DIS
LIN {X 101.7885,Y 100.3867,Z 190,A 44.8958,B 1.3167,C -0.0025,E1 1.4342,E2 409.5098} C_DIS
LIN {X 98.6524,Y 103.4696,Z 190,A 46.5039,B 1.3167,C -0.0054,E1 1.431,E2 407.9209} C_DIS
LIN {X 95.9178,Y 106.0097,Z 190,A 47.8749,B 1.3167,C -0.0078,E1 1.4282,E2 406.5655} C_DIS
LIN {X 92.7135,Y 108.8231,Z 190,A 49.4783,B 1.3167,C -0.0107,E1 1.4248,E2 404.9752} C_DIS
LIN {X 89.9304,Y 111.1342,Z 190,A 50.9106,B 1.3167,C -0.0135,E1 1.4217,E2 403.5451} C_DIS
LIN {X 86.4725,Y 113.8461,Z 190,A 52.5704,B 1.3167,C -0.0163,E1 1.418,E2 401.8979} C_DIS
LIN {X 82.9799,Y 116.4157,Z 190,A 54.0817,B 1.3167,C -0.0184,E1 1.4147,E2 400.4147} C_DIS
LIN {X 79.4275,Y 118.8676,Z 190,A 55.6908,B 1.3167,C -0.0209,E1 1.411,E2 398.8207} C_DIS
LIN {X 76.0875,Y 121.033,Z 190,A 57.2323,B 1.3166,C -0.0234,E1 1.4073,E2 397.2859} C_DIS
LIN {X 72.7455,Y 123.0711,Z 190,A 58.6833,B 1.3166,C -0.0255,E1 1.4039,E2 395.8496} C_DIS
LIN {X 69.0395,Y 125.1872,Z 190,A 60.3005,B 1.3165,C -0.0278,E1 1.4,E2 394.244} C_DIS
LIN {X 65.7292,Y 126.9567,Z 190,A 61.8371,B 1.3165,C -0.0303,E1 1.3961,E2 392.7036} C_DIS
LIN {X 61.9124,Y 128.8589,Z 190,A 63.339,B 1.3164,C -0.0319,E1 1.3924,E2 391.2272} C_DIS
LIN {X 58.6245,Y 130.3875,Z 190,A 64.777,B 1.3164,C -0.0339,E1 1.3887,E2 389.7913} C_DIS
LIN {X 54.4968,Y 132.1673,Z 190,A 66.4007,B 1.3164,C -0.0355,E1 1.3846,E2 388.1896} C_DIS
LIN {X 51.2391,Y 133.4638,Z 190,A 67.7228,B 1.3163,C -0.037,E1 1.3812,E2 386.8778} C_DIS
LIN {X 48.1552,Y 134.6064,Z 190,A 69.1108,B 1.3163,C -0.0389,E1 1.3775,E2 385.4815} C_DIS
LIN {X 43.3634,Y 136.2253,Z 190,A 70.9839,B 1.3162,C -0.0406,E1 1.3725,E2 383.6276} C_DIS
LIN {X 39.58,Y 137.3736,Z 190,A 72.452,B 1.3162,C -0.0419,E1 1.3686,E2 382.174} C_DIS
LIN {X 36.2062,Y 138.3013,Z 190,A 73.7991,B 1.3161,C -0.0431,E1 1.365,E2 380.834} C_DIS
LIN {X 32.811,Y 139.1462,Z 190,A 75.1495,B 1.3161,C -0.0443,E1 1.3613,E2 379.4902} C_DIS
LIN {X 29.3803,Y 139.9114,Z 190,A 76.5124,B 1.3161,C -0.0454,E1 1.3576,E2 378.1333} C_DIS
LIN {X 26.1579,Y 140.5489,Z 190,A 77.8317,B 1.316,C -0.0465,E1 1.3539,E2 376.8139} C_DIS
LIN {X 22.328,Y 141.2071,Z 190,A 79.2697,B 1.316,C -0.0472,E1 1.35,E2 375.3907} C_DIS
LIN {X 19.2388,Y 141.6619,Z 190,A 80.5337,B 1.316,C -0.0482,E1 1.3465,E2 374.1256} C_DIS
LIN {X 15.4077,Y 142.1281,Z 190,A 82.0123,B 1.3159,C -0.0489,E1 1.3423,E2 372.6558} C_DIS
LIN {X 12.0272,Y 142.454,Z 190,A 83.361,B 1.3159,C -0.0497,E1 1.3386,E2 371.309} C_DIS
LIN {X 8.7591,Y 142.6923,Z 190,A 84.6766,B 1.3159,C -0.0503,E1 1.3349,E2 369.9936} C_DIS
LIN {X 5.031,Y 142.8734,Z 190,A 86.1022,B 1.3159,C -0.0508,E1 1.3309,E2 368.5769} C_DIS
LIN {X 1.5265,Y 142.9547,Z 190,A 87.4594,B 1.3158,C -0.0512,E1 1.3271,E2 367.2261} C_DIS
LIN {X -1.7576,Y 142.9515,Z 190,A 88.8271,B 1.3158,C -0.0517,E1 1.3232,E2 365.8526} C_DIS
LIN {X -5.7098,Y 142.8469,Z 190,A 90.3415,B 1.3158,C -0.0519,E1 1.319,E2 364.3473} C_DIS
LIN {X -8.7718,Y 142.6915,Z 190,A 91.5965,B 1.3158,C -0.0522,E1 1.3155,E2 363.0896} C_DIS
LIN {X -12.2667,Y 142.4338,Z 190,A 93.0261,B 1.3158,C -0.0524,E1 1.3115,E2 361.6577} C_DIS
LIN {X -16.0013,Y 142.0642,Z 190,A 94.4829,B 1.3158,C -0.0524,E1 1.3074,E2 360.2073} C_DIS
LIN {X -19.2547,Y 141.6598,Z 190,A 95.8006,B 1.3158,C -0.0523,E1 1.3037,E2 358.8897} C_DIS
LIN {X -22.7188,Y 141.1463,Z 190,A 97.3004,B 1.3158,C -0.0524,E1 1.2995,E2 357.379} C_DIS
LIN {X -26.17,Y 140.5466,Z 190,A 98.7079,B 1.3158,C -0.0522,E1 1.2956,E2 355.9717} C_DIS
LIN {X -29.8644,Y 139.8068,Z 190,A 100.2317,B 1.3158,C -0.0518,E1 1.2914,E2 354.447} C_DIS
LIN {X -33.7634,Y 138.9167,Z 190,A 101.6191,B 1.3158,C -0.0508,E1 1.2877,E2 353.086} C_DIS
LIN {X -36.4202,Y 138.2442,Z 190,A 102.9008,B 1.3158,C -0.0508,E1 1.2842,E2 351.7831} C_DIS
LIN {X -40.1505,Y 137.2066,Z 190,A 104.4589,B 1.3158,C -0.0501,E1 1.2799,E2 350.225} C_DIS
LIN {X -43.4056,Y 136.2118,Z 190,A 105.8711,B 1.3158,C -0.0495,E1 1.2761,E2 348.8078} C_DIS
LIN {X -46.7315,Y 135.1069,Z 190,A 107.3087,B 1.3158,C -0.0488,E1 1.2723,E2 347.367} C_DIS
LIN {X -49.8154,Y 134.0009,Z 190,A 108.655,B 1.3159,C -0.048,E1 1.2687,E2 346.0174} C_DIS
LIN {X -53.0839,Y 132.7401,Z 190,A 110.1581,B 1.3159,C -0.0471,E1 1.2648,E2 344.5032} C_DIS
LIN {X -56.5451,Y 131.3026,Z 190,A 111.7467,B 1.3159,C -0.0461,E1 1.2606,E2 342.905} C_DIS
LIN {X -60.2546,Y 129.6423,Z 190,A 113.327,B 1.316,C -0.0446,E1 1.2566,E2 341.3314} C_DIS
LIN {X -63.2566,Y 128.204,Z 190,A 114.5344,B 1.316,C -0.0431,E1 1.2536,E2 340.1401} C_DIS
LIN {X -65.8267,Y 126.9055,Z 190,A 115.9147,B 1.3161,C -0.0423,E1 1.2501,E2 338.7333} C_DIS
LIN {X -69.0517,Y 125.1805,Z 190,A 117.5693,B 1.3161,C -0.0411,E1 1.2459,E2 337.0568} C_DIS
LIN {X -72.7552,Y 123.0653,Z 190,A 119.2483,B 1.3162,C -0.0391,E1 1.2419,E2 335.3825} C_DIS
LIN {X -75.8453,Y 121.1852,Z 190,A 120.77,B 1.3162,C -0.0374,E1 1.2382,E2 333.853} C_DIS
LIN {X -78.7912,Y 119.2905,Z 190,A 122.3668,B 1.3162,C -0.0359,E1 1.2344,E2 332.2336} C_DIS
LIN {X -82.4313,Y 116.8046,Z 190,A 124.2471,B 1.3164,C -0.0336,E1 1.23,E2 330.3406} C_DIS
LIN {X -85.8719,Y 114.2994,Z 190,A 125.9078,B 1.3164,C -0.0311,E1 1.2263,E2 328.6864} C_DIS
LIN {X -89.1042,Y 111.7975,Z 190,A 127.7042,B 1.3164,C -0.0288,E1 1.2223,E2 326.8717} C_DIS
LIN {X -92.0426,Y 109.3912,Z 190,A 129.2808,B 1.3165,C -0.0265,E1 1.2189,E2 325.2895} C_DIS
LIN {X -95.2657,Y 106.596,Z 190,A 131.1549,B 1.3165,C -0.0238,E1 1.2149,E2 323.3964} C_DIS
LIN {X -98.0293,Y 104.0601,Z 190,A 132.826,B 1.3166,C -0.0214,E1 1.2114,E2 321.7056} C_DIS
LIN {X -101.1721,Y 101.0077,Z 190,A 134.5953,B 1.3166,C -0.0182,E1 1.2079,E2 319.9359} C_DIS
LIN {X -104.1411,Y 97.9434,Z 190,A 136.4541,B 1.3166,C -0.0152,E1 1.2043,E2 318.0597} C_DIS
LIN {X -106.5991,Y 95.2622,Z 190,A 138.1725,B 1.3167,C -0.0126,E1 1.201,E2 316.3101} C_DIS
LIN {X -109.4677,Y 91.9514,Z 190,A 139.9227,B 1.3167,C -0.0091,E1 1.1978,E2 314.5617} C_DIS
LIN {X -112.0915,Y 88.7348,Z 190,A 141.7539,B 1.3167,C -0.0058,E1 1.1945,E2 312.7108} C_DIS
LIN {X -114.3876,Y 85.7549,Z 190,A 143.538,B 1.3167,C -0.0028,E1 1.1915,E2 310.8932} C_DIS
LIN {X -116.9602,Y 82.2107,Z 190,A 145.2957,B 1.3167,C 0.001,E1 1.1886,E2 309.1363} C_DIS
LIN {X -119.3582,Y 78.6883,Z 190,A 147.1845,B 1.3167,C 0.0047,E1 1.1856,E2 307.2259} C_DIS
LIN {X -121.2482,Y 75.7442,Z 190,A 148.7242,B 1.3167,C 0.0079,E1 1.1833,E2 305.6699} C_DIS
LIN {X -123.4517,Y 72.0976,Z 190,A 150.6209,B 1.3167,C 0.0117,E1 1.1805,E2 303.7505} C_DIS
LIN {X -125.6101,Y 68.2671,Z 190,A 152.606,B 1.3167,C 0.0159,E1 1.1778,E2 301.7382} C_DIS
LIN {X -127.3,Y 65.057,Z 190,A 154.0999,B 1.3167,C 0.0194,E1 1.1759,E2 300.2401} C_DIS
LIN {X -128.871,Y 61.8871,Z 190,A 155.6858,B 1.3166,C 0.0228,E1 1.1739,E2 298.6338} C_DIS
LIN {X -130.3882,Y 58.6231,Z 190,A 157.3989,B 1.3166,C 0.0263,E1 1.1719,E2 296.887} C_DIS
LIN {X -132.1697,Y 54.491,Z 190,A 159.2941,B 1.3164,C 0.0309,E1 1.1698,E2 294.9813} C_DIS
LIN {X -133.4771,Y 51.205,Z 190,A 160.8495,B 1.3164,C 0.0345,E1 1.1682,E2 293.409} C_DIS
LIN {X -134.6019,Y 48.1676,Z 190,A 162.3094,B 1.3162,C 0.0379,E1 1.1668,E2 291.929} C_DIS
LIN {X -135.7412,Y 44.8568,Z 190,A 163.8745,B 1.3162,C 0.0415,E1 1.1654,E2 290.3439} C_DIS
LIN {X -136.873,Y 41.2774,Z 190,A 165.548,B 1.316,C 0.0455,E1 1.164,E2 288.6495} C_DIS
LIN {X -137.8577,Y 37.8603,Z 190,A 167.1371,B 1.3159,C 0.0493,E1 1.1628,E2 287.0399} C_DIS
LIN {X -138.7437,Y 34.4737,Z 190,A 168.7029,B 1.3157,C 0.0531,E1 1.1617,E2 285.4537} C_DIS
LIN {X -139.5453,Y 31.0717,Z 190,A 170.2669,B 1.3156,C 0.0569,E1 1.1607,E2 283.8692} C_DIS
LIN {X -140.2628,Y 27.6544,Z 190,A 171.9321,B 1.3154,C 0.0608,E1 1.1598,E2 282.17} C_DIS
LIN {X -140.9135,Y 24.1141,Z 190,A 173.4406,B 1.3152,C 0.0647,E1 1.159,E2 280.6537} C_DIS
LIN {X -141.4504,Y 20.7323,Z 190,A 174.9319,B 1.315,C 0.0685,E1 1.1584,E2 279.1475} C_DIS
LIN {X -141.8884,Y 17.4859,Z 190,A 176.4789,B 1.3148,C 0.0722,E1 1.1578,E2 277.5702} C_DIS
LIN {X -142.2953,Y 13.7785,Z 190,A 178.1449,B 1.3146,C 0.0763,E1 1.1573,E2 275.8822} C_DIS
LIN {X -142.5901,Y 10.2902,Z 190,A 179.6732,B 1.3143,C 0.0803,E1 1.157,E2 274.3381} C_DIS
LIN {X -142.8006,Y 6.7793,Z 190,A -178.7156,B 1.3141,C 0.0842,E1 1.1568,E2 272.7007} C_DIS
LIN {X -142.925,Y 3.2796,Z 190,A -177.1056,B 1.3138,C 0.0882,E1 1.1566,E2 271.0638} C_DIS
LIN {X -142.963,Y -0.0079,Z 190,A -175.6201,B 1.3136,C 0.0919,E1 1.1566,E2 269.5564} C_DIS
LIN {X -142.9186,Y -3.5101,Z 190,A -174.0566,B 1.3133,C 0.0958,E1 1.1566,E2 267.972} C_DIS
LIN {X -142.7757,Y -7.2746,Z 190,A -172.4192,B 1.313,C 0.1,E1 1.1569,E2 266.3181} C_DIS
LIN {X -142.5715,Y -10.5449,Z 190,A -170.908,B 1.3127,C 0.1037,E1 1.1572,E2 264.7806} C_DIS
LIN {X -142.2498,Y -14.2529,Z 190,A -169.2457,B 1.3124,C 0.1078,E1 1.1576,E2 263.0959} C_DIS
LIN {X -141.8593,Y -17.7302,Z 190,A -167.6774,B 1.312,C 0.1117,E1 1.1581,E2 261.5057} C_DIS
LIN {X -141.4106,Y -21.0103,Z 190,A -166.1735,B 1.3117,C 0.1154,E1 1.1587,E2 259.9781} C_DIS
LIN {X -140.8156,Y -24.6774,Z 190,A -164.5732,B 1.3114,C 0.1194,E1 1.1595,E2 258.3632} C_DIS
LIN {X -140.2179,Y -27.8763,Z 190,A -163.0413,B 1.311,C 0.123,E1 1.1603,E2 256.8005} C_DIS
LIN {X -139.4887,Y -31.3197,Z 190,A -161.4081,B 1.3107,C 0.1268,E1 1.1613,E2 255.1371} C_DIS
LIN {X -138.6756,Y -34.7419,Z 190,A -159.8905,B 1.3103,C 0.1305,E1 1.1623,E2 253.6052} C_DIS
LIN {X -137.7818,Y -38.1317,Z 190,A -158.3246,B 1.3099,C 0.1343,E1 1.1635,E2 252.0174} C_DIS
LIN {X -136.7383,Y -41.7175,Z 190,A -156.6578,B 1.3095,C 0.1382,E1 1.1648,E2 250.3275} C_DIS
LIN {X -135.6682,Y -45.076,Z 190,A -155.0854,B 1.3091,C 0.1418,E1 1.1662,E2 248.7334} C_DIS
LIN {X -134.5229,Y -48.3867,Z 190,A -153.554,B 1.3087,C 0.1454,E1 1.1677,E2 247.1846} C_DIS
LIN {X -133.38,Y -51.4547,Z 190,A -152.0697,B 1.3084,C 0.1487,E1 1.1692,E2 245.6767} C_DIS
LIN {X -131.9719,Y -54.9647,Z 190,A -150.3919,B 1.3079,C 0.1525,E1 1.171,E2 243.9765} C_DIS
LIN {X -130.3339,Y -58.7445,Z 190,A -148.4369,B 1.3075,C 0.1565,E1 1.1732,E2 241.979} C_DIS
LIN {X -128.4255,Y -62.8075,Z 190,A -146.4512,B 1.3069,C 0.1607,E1 1.1757,E2 239.9674} C_DIS
LIN {X -126.8931,Y -65.8503,Z 190,A -145.0897,B 1.3065,C 0.164,E1 1.1774,E2 238.6069} C_DIS
LIN {X -125.1868,Y -69.0403,Z 190,A -143.3489,B 1.3061,C 0.1673,E1 1.1798,E2 236.825} C_DIS
LIN {X -123.0715,Y -72.7447,Z 190,A -141.5397,B 1.3056,C 0.1711,E1 1.1823,E2 235.0021} C_DIS
LIN {X -120.7635,Y -76.5145,Z 190,A -139.6339,B 1.3051,C 0.175,E1 1.1852,E2 233.0775} C_DIS
LIN {X -118.3781,Y -80.1552,Z 190,A -137.7442,B 1.3046,C 0.1787,E1 1.1881,E2 231.1673} C_DIS
LIN {X -116.0694,Y -83.4642,Z 190,A -135.9004,B 1.3041,C 0.182,E1 1.1912,E2 229.2912} C_DIS
LIN {X -113.6948,Y -86.6706,Z 190,A -134.2469,B 1.3037,C 0.1853,E1 1.194,E2 227.63} C_DIS
LIN {X -111.1343,Y -89.9302,Z 190,A -132.3574,B 1.3032,C 0.1884,E1 1.1973,E2 225.7077} C_DIS
LIN {X -108.0428,Y -93.6225,Z 190,A -130.2266,B 1.3027,C 0.192,E1 1.2013,E2 223.5481} C_DIS
LIN {X -105.2576,Y -96.7423,Z 190,A -128.5421,B 1.3023,C 0.1951,E1 1.2044,E2 221.8626} C_DIS
LIN {X -102.3892,Y -99.7742,Z 190,A -126.6881,B 1.3018,C 0.1979,E1 1.2081,E2 219.9824} C_DIS
LIN {X -99.75,Y -102.4126,Z 190,A -124.9822,B 1.3015,C 0.2003,E1 1.2116,E2 218.2458} C_DIS
LIN {X -96.0901,Y -105.8533,Z 190,A -122.9407,B 1.301,C 0.2036,E1 1.2158,E2 216.2002} C_DIS
LIN {X -92.7194,Y -108.8181,Z 190,A -121.039,B 1.3005,C 0.2063,E1 1.2198,E2 214.2835} C_DIS
LIN {X -89.9233,Y -111.1399,Z 190,A -119.3992,B 1.3002,C 0.2083,E1 1.2235,E2 212.6168} C_DIS
LIN {X -86.4619,Y -113.8541,Z 190,A -117.5138,B 1.2998,C 0.2106,E1 1.2277,E2 210.7133} C_DIS
LIN {X -83.0331,Y -116.3776,Z 190,A -115.8232,B 1.2994,C 0.213,E1 1.2315,E2 209.0249} C_DIS
LIN {X -80.0558,Y -118.4454,Z 190,A -114.198,B 1.2992,C 0.2146,E1 1.2354,E2 207.3742} C_DIS
LIN {X -76.4855,Y -120.7818,Z 190,A -112.4947,B 1.2988,C 0.2167,E1 1.2394,E2 205.6717} C_DIS
LIN {X -73.4029,Y -122.6797,Z 190,A -110.8833,B 1.2986,C 0.2181,E1 1.2433,E2 204.0364} C_DIS
LIN {X -69.322,Y -125.0308,Z 190,A -108.9379,B 1.2983,C 0.22,E1 1.2481,E2 202.0821} C_DIS
LIN {X -65.7336,Y -126.9544,Z 190,A -107.1727,B 1.2981,C 0.2213,E1 1.2525,E2 200.2968} C_DIS
LIN {X -61.9094,Y -128.8603,Z 190,A -105.5574,B 1.2977,C 0.2231,E1 1.2566,E2 198.6956} C_DIS
LIN {X -58.6279,Y -130.386,Z 190,A -103.9558,B 1.2976,C 0.224,E1 1.2607,E2 197.0712} C_DIS
LIN {X -54.4991,Y -132.1663,Z 190,A -102.1937,B 1.2973,C 0.2255,E1 1.2653,E2 195.3147} C_DIS
LIN {X -51.2322,Y -133.4665,Z 190,A -100.6393,B 1.2973,C 0.2261,E1 1.2694,E2 193.7383} C_DIS
LIN {X -46.6954,Y -135.1194,Z 190,A -98.7091,B 1.297,C 0.2273,E1 1.2745,E2 191.8083} C_DIS
LIN {X -43.153,Y -136.2925,Z 190,A -97.2213,B 1.2969,C 0.2281,E1 1.2785,E2 190.3213} C_DIS
LIN {X -39.5891,Y -137.371,Z 190,A -95.7194,B 1.2968,C 0.2287,E1 1.2826,E2 188.8175} C_DIS
LIN {X -36.2149,Y -138.299,Z 190,A -94.3022,B 1.2967,C 0.2292,E1 1.2864,E2 187.3976} C_DIS
LIN {X -32.8046,Y -139.1478,Z 190,A -92.8791,B 1.2967,C 0.2296,E1 1.2903,E2 185.9718} C_DIS
LIN {X -29.3782,Y -139.9118,Z 190,A -91.4559,B 1.2966,C 0.2299,E1 1.2942,E2 184.5457} C_DIS
LIN {X -25.7502,Y -140.6236,Z 190,A -90.0112,B 1.2965,C 0.2303,E1 1.2982,E2 183.1059} C_DIS
LIN {X -22.4833,Y -141.183,Z 190,A -88.6173,B 1.2965,C 0.2303,E1 1.3021,E2 181.7017} C_DIS
LIN {X -19.2427,Y -141.6614,Z 190,A -87.2956,B 1.2965,C 0.2303,E1 1.3058,E2 180.3781} C_DIS
LIN {X -15.7474,Y -142.0916,Z 190,A -85.8451,B 1.2965,C 0.2301,E1 1.3099,E2 178.9211} C_DIS
LIN {X -12.0307,Y -142.4537,Z 190,A -84.4124,B 1.2965,C 0.2301,E1 1.3139,E2 177.4973} C_DIS
LIN {X -8.7637,Y -142.692,Z 190,A -83.0797,B 1.2965,C 0.2299,E1 1.3176,E2 176.161} C_DIS
LIN {X -5.034,Y -142.8732,Z 190,A -81.5241,B 1.2967,C 0.2293,E1 1.322,E2 174.5958} C_DIS
LIN {X -1.5228,Y -142.9547,Z 190,A -80.2766,B 1.2967,C 0.2295,E1 1.3255,E2 173.3716} C_DIS
LIN {X 1.0342,Y -142.9562,Z 190,A -79.5486,B 1.2965,C 0.2302,E1 1.3274,E2 172.6873} C_DIS
Enddeposition()
LIN {X 0.97,Y -133.9818,Z 191,A -77.9723,B 1.0089,C 0.2063,E1 1.0433,E2 170.7026} C_DIS
Startdeposition()
$VEL.CP = VEL_PRINT
LIN {X -1.3193,Y -133.9827,Z 191,A -79.3559,B 1.0086,C 0.2079,E1 1.0393,E2 172.1436} C_DIS
LIN {X -4.9338,Y -133.8974,Z 191,A -80.8062,B 1.0086,C 0.2082,E1 1.0352,E2 173.5812} C_DIS
LIN {X -8.2125,Y -133.736,Z 191,A -82.1189,B 1.0086,C 0.2083,E1 1.0315,E2 174.8819} C_DIS
LIN {X -11.1705,Y -133.5214,Z 191,A -83.4397,B 1.0084,C 0.2088,E1 1.0278,E2 176.2107} C_DIS
LIN {X -14.776,Y -133.1713,Z 191,A -84.9346,B 1.0084,C 0.2088,E1 1.0236,E2 177.6988} C_DIS
LIN {X -17.6989,Y -132.814,Z 191,A -86.2524,B 1.0084,C 0.2091,E1 1.0199,E2 179.0254} C_DIS
LIN {X -20.9474,Y -132.3409,Z 191,A -87.6235,B 1.0084,C 0.2091,E1 1.0161,E2 180.3925} C_DIS
LIN {X -24.5284,Y -131.725,Z 191,A -89.1968,B 1.0084,C 0.2091,E1 1.0117,E2 181.9692} C_DIS
LIN {X -27.1032,Y -131.2184,Z 191,A -90.4367,B 1.0084,C 0.2091,E1 1.0082,E2 183.226} C_DIS
LIN {X -30.3456,Y -130.5071,Z 191,A -91.8786,B 1.0084,C 0.209,E1 1.0042,E2 184.6716} C_DIS
LIN {X -34.149,Y -129.5634,Z 191,A -93.4494,B 1.0085,C 0.2083,E1 0.9999,E2 186.2283} C_DIS
LIN {X -37.3152,Y -128.6871,Z 191,A -94.8767,B 1.0086,C 0.2079,E1 0.9961,E2 187.6593} C_DIS
LIN {X -40.1345,Y -127.8371,Z 191,A -96.164,B 1.0087,C 0.2075,E1 0.9926,E2 188.951} C_DIS
LIN {X -43.6031,Y -126.6945,Z 191,A -97.758,B 1.0088,C 0.2068,E1 0.9883,E2 190.5499} C_DIS
LIN {X -47.5312,Y -125.2747,Z 191,A -99.7558,B 1.009,C 0.2062,E1 0.9829,E2 192.5778} C_DIS
LIN {X -51.2784,Y -123.7873,Z 191,A -101.2462,B 1.0093,C 0.2047,E1 0.9791,E2 194.036} C_DIS
LIN {X -53.8776,Y -122.6801,Z 191,A -102.7497,B 1.0093,C 0.2043,E1 0.9751,E2 195.5812} C_DIS
LIN {X -56.9697,Y -121.2754,Z 191,A -104.1453,B 1.0096,C 0.2031,E1 0.9715,E2 196.9692} C_DIS
LIN {X -59.9364,Y -119.8365,Z 191,A -105.6177,B 1.0098,C 0.202,E1 0.9678,E2 198.4506} C_DIS
LIN {X -62.7341,Y -118.3946,Z 191,A -107.0814,B 1.01,C 0.201,E1 0.9641,E2 199.9308} C_DIS
LIN {X -66.059,Y -116.5741,Z 191,A -108.7207,B 1.0103,C 0.1994,E1 0.96,E2 201.573} C_DIS
LIN {X -68.638,Y -115.0738,Z 191,A -110.1215,B 1.0106,C 0.1982,E1 0.9566,E2 202.9913} C_DIS
LIN {X -71.6857,Y -113.2005,Z 191,A -111.6207,B 1.0109,C 0.1965,E1 0.953,E2 204.4865} C_DIS
LIN {X -74.7175,Y -111.2232,Z 191,A -113.4966,B 1.0112,C 0.195,E1 0.9485,E2 206.408} C_DIS
LIN {X -78.2119,Y -108.7942,Z 191,A -115.2855,B 1.0116,C 0.1927,E1 0.9444,E2 208.1928} C_DIS
Enddeposition()
END
